// TwinCAT 3 PLC project tmo_optics
// Title: lcls-plc-tmo-optics
// Company: SLAC
// ProjectVersion: 0.0.0
// ProgramVersion: 3.1.4026.17
// CompilerDefines: K
// libraries:
//   LCLS General, * (SLAC)
//   lcls-twincat-common-components, * (SLAC)
//   lcls-twincat-optics, * (SLAC)
//   Tc2_MC2, * (Beckhoff Automation GmbH)
//   Tc2_SerialCom, * (Beckhoff Automation GmbH)
//   Tc2_Standard, * (Beckhoff Automation GmbH)
//   Tc2_System, * (Beckhoff Automation GmbH)
//   Tc2_Utilities, * (Beckhoff Automation GmbH)
//   Tc3_Module, * (Beckhoff Automation GmbH)
//   TcUnit, * (www.tcunit.org)
//   lcls-twincat-motion,4.4.0,SLAC
//   PMPS,3.12.0,SLAC - LCLS
// project tree:
//   DUTs/ ENUM_Si_B4C_Coating_States.TcDUT, ENUM_Si_B4C_Coating_States_1D.TcDUT, E_HomeState.TcDUT (not stored)
//   GVLs/ GVL_COM_Buffers.TcGVL (not stored), GVL_M1K4.TcGVL (not stored), GVL_M1K4_Constants.TcGVL (not stored), GVL_M2K4_RTD.TcGVL (not stored), GVL_M2K4_Constants.TcGVL (not stored), GVL_M3K4_RTD.TcGVL (not stored), GVL_M3K4_Constants.TcGVL (not stored), GVL_M4K4_RTD.TcGVL (not stored), GVL_M5K4_RTD.TcGVL (not stored), GVL_PMPS.TcGVL, GVL_SerialIO.TcGVL (not stored)
//   / PiezoDriver.TcTTO (not stored), PlcTask.TcTTO (not stored), SerialIO.TcTTO (not stored)
//   POUs/ FB_Offset_Coating_States.TcPOU (not stored), FB_KBO_Coating_States.TcPOU (not stored), Main.TcPOU, PRG_1_PlcTask.TcPOU (not stored), PRG_Environment.TcPOU (not stored), PRG_MR1K4_SOMS.TcPOU (not stored), PRG_MR2K4_KBO.TcPOU (not stored), PRG_MR3K4_KBO.TcPOU (not stored), PRG_MR4K4_KBO.TcPOU (not stored), PRG_MR5K4_KBO.TcPOU (not stored), PRG_PMPS.TcPOU, PRG_SL2K4_SCATTER.TcPOU (not stored), PRG_States.TcPOU, P_StripeProtections.TcPOU (not stored)
//   POUs/Serial Comm/ PiezoSerial.TcPOU (not stored), P_Serial_Com.TcPOU (not stored)
//   POUs/temp/ FB_SLITS.TcPOU (not stored)
// real-time tasks:
//   TASK PlcTask: cycle T#10ms, priority 20, ADS port 350
//   TASK PiezoDriver: cycle T#1ms, priority 3, ADS port 351
//   TASK SerialIO: cycle T#2ms, priority 1, ADS port 352
// motion (NC):
//   TASK NC-Task 1 SAF: cycle T#2ms, priority 4, ADS port 501
//   TASK NC-Task 1 SVB: cycle T#10ms, priority 8, ADS port 511
//   AXIS M1K4-Yup (id 1)
//   AXIS M1K4-Ydwn (id 2)
//   AXIS M1K4-Xup (id 3)
//   AXIS M1K4-Xdwn (id 4)
//   AXIS M1K4-Pitch (id 5)
//   AXIS M1K4-Bender (id 6)
//   AXIS M2K4-X (id 7)
//   AXIS M2K4-Y (id 8)
//   AXIS M2K4-rY (id 9)
//   AXIS M2K4-BEND-US (id 10)
//   AXIS M2K4-BEND-DS (id 11)
//   AXIS M3K4-X (id 12)
//   AXIS M3K4-Y (id 13)
//   AXIS M3K4-rX (id 14)
//   AXIS M3K4-BEND-US (id 15)
//   AXIS M3K4-BEND-DS (id 16)
//   AXIS M4K4 X (id 17)
//     Dynamic: AccelerationMaximum=100, DecelerationMaximum=100, Acceleration=100, Deceleration=100, DelayTime=0.008
//     Velo: Maximum=0.3
//     OtherSettings: AllowMotionCmdToSlave=true
//     encoder EncType=29
//       EncPara: ScaleFactorNumerator=5e-06, Offset=-28.961399, MaxCount=#xffffffff
//         SoftEndMinControl: Enable=true, Range=-11.4
//         SoftEndMaxControl: Enable=true, Range=13.4
//         Inc: RefSoftSyncMask=#x0000ffff
//     drive DrvType=24
//       DrvPara: Inverse=true
//         Analog: VeloReferenz=20, ScaleFactorActTorque=0.1
//         TimeComp: TaskDelayCycles=1
//     controller CtrType=2
//       CtrPara: PriorControlFactor=1
//         PosDiffControl: Range=0.2
//         PID: DeadBandPosition=0.001
//         Observer: BandWidth=20
//   AXIS M4K4 Y (id 18)
//     Dynamic: AccelerationMaximum=100, DecelerationMaximum=100, Acceleration=100, Deceleration=100, DelayTime=0.008
//     Velo: Maximum=0.2
//     OtherSettings: AllowMotionCmdToSlave=true
//     encoder EncType=29
//       EncPara: ScaleFactorNumerator=5e-06, Offset=-30.3992, MaxCount=#xffffffff
//         SoftEndMinControl: Enable=true, Range=-2.2
//         SoftEndMaxControl: Enable=true, Range=2.3
//         Inc: RefSoftSyncMask=#x0000ffff
//     drive DrvType=24
//       DrvPara: Inverse=true
//         Analog: VeloReferenz=1.25, ScaleFactorActTorque=0.1
//         TimeComp: TaskDelayCycles=1
//     controller CtrType=2
//       CtrPara: PriorControlFactor=1
//         PosDiffControl: Range=0.2
//         PID: PosKp=3, DeadBandPosition=0.001
//         Observer: BandWidth=20
//   AXIS M4K4 Z (id 19)
//     Dynamic: AccelerationMaximum=100, DecelerationMaximum=100, Acceleration=100, Deceleration=100, DelayTime=0.008
//     Velo: Maximum=0.2
//     OtherSettings: AllowMotionCmdToSlave=true
//     encoder EncType=29
//       EncPara: ScaleFactorNumerator=5e-06, Offset=-21445.3535, MaxCount=#xffffffff
//         SoftEndMinControl: Enable=true, Range=-1.5
//         SoftEndMaxControl: Enable=true, Range=0.85
//         Inc: RefSoftSyncMask=#x0000ffff
//     drive DrvType=24
//       DrvPara: Inverse=true
//         Analog: VeloReferenz=1.25, ScaleFactorActTorque=0.1
//         TimeComp: TaskDelayCycles=1
//     controller CtrType=2
//       CtrPara: PriorControlFactor=1
//         PosDiffControl: Range=0.2
//         PID: PosKp=2, DeadBandPosition=0.01
//         Observer: BandWidth=20
//   AXIS M4K4 rX (id 20)
//     General: UnitName=urad
//     Dynamic: AccelerationMaximum=100, DecelerationMaximum=100, Acceleration=100, Deceleration=100, DelayTime=0.008
//     Velo: Maximum=50
//     OtherSettings: AllowMotionCmdToSlave=true
//     encoder EncType=29
//       EncPara: ScaleFactorNumerator=0.0025826, Offset=-132192.8499, MaxCount=#xffffffff
//         FilterTime: TPos=0.2
//         SoftEndMinControl: Enable=true, Range=-500
//         SoftEndMaxControl: Enable=true, Range=500
//         Inc: RefSoftSyncMask=#x0000ffff
//     drive DrvType=24
//       Analog: VeloReferenz=140.69, ScaleFactorActTorque=0.1
//       TimeComp: TaskDelayCycles=1
//     controller CtrType=2
//       CtrPara: PriorControlFactor=1
//         PosDiffControl: Range=10
//         PID: PosExtKp=4, DeadBandPosition=0.01
//         Observer: BandWidth=20
//   AXIS M5K4 X (id 21)
//     Dynamic: AccelerationMaximum=100, DecelerationMaximum=100, Acceleration=100, Deceleration=100, DelayTime=0.008
//     Velo: Maximum=0.2
//     OtherSettings: AllowMotionCmdToSlave=true
//     encoder EncType=29
//       EncPara: ScaleFactorNumerator=5e-06, Offset=-29.80379, MaxCount=#xffffffff
//         SoftEndMinControl: Enable=true, Range=-2.1
//         SoftEndMaxControl: Enable=true, Range=2.6
//         Inc: RefSoftSyncMask=#x0000ffff
//     drive DrvType=24
//       DrvPara: Inverse=true
//         Analog: VeloReferenz=20, ScaleFactorActTorque=0.1
//         TimeComp: TaskDelayCycles=1
//     controller CtrType=2
//       CtrPara: PriorControlFactor=1
//         PosDiffControl: Range=0.2
//         PID: DeadBandPosition=0.001
//         Observer: BandWidth=20
//   AXIS M5K4 Y (id 22)
//     Dynamic: AccelerationMaximum=100, DecelerationMaximum=100, Acceleration=100, Deceleration=100, DelayTime=0.008
//     Velo: Maximum=0.3
//     OtherSettings: AllowMotionCmdToSlave=true
//     encoder EncType=29
//       EncPara: ScaleFactorNumerator=5e-06, Offset=-29.7766, MaxCount=#xffffffff
//         SoftEndMinControl: Enable=true, Range=-12.3
//         SoftEndMaxControl: Enable=true, Range=12.33
//         Inc: RefSoftSyncMask=#x0000ffff
//     drive DrvType=24
//       DrvPara: Inverse=true
//         Analog: VeloReferenz=1.25, ScaleFactorActTorque=0.1
//         TimeComp: TaskDelayCycles=1
//     controller CtrType=2
//       CtrPara: PriorControlFactor=1
//         PosDiffControl: Range=0.2
//         PID: DeadBandPosition=0.001
//         Observer: BandWidth=20
//   AXIS M5K4 Z (id 23)
//     Dynamic: AccelerationMaximum=100, DecelerationMaximum=100, Acceleration=100, Deceleration=100, DelayTime=0.008
//     Velo: Maximum=0.2
//     OtherSettings: AllowMotionCmdToSlave=true
//     encoder EncType=29
//       EncPara: ScaleFactorNumerator=5e-06, Offset=-21444.5039, MaxCount=#xffffffff
//         SoftEndMinControl: Enable=true, Range=-0.69
//         SoftEndMaxControl: Enable=true, Range=1.02
//         Inc: RefSoftSyncMask=#x0000ffff
//     drive DrvType=24
//       DrvPara: Inverse=true
//         Analog: VeloReferenz=1.25, ScaleFactorActTorque=0.1
//         TimeComp: TaskDelayCycles=1
//     controller CtrType=2
//       CtrPara: PriorControlFactor=1
//         PosDiffControl: Range=0.2
//         PID: PosExtVelo=1, DeadBandPosition=0.01
//         Observer: BandWidth=20
//   AXIS M5K4 rY (id 24)
//     General: UnitName=urad
//     Dynamic: AccelerationMaximum=100, DecelerationMaximum=100, Acceleration=100, Deceleration=100, DelayTime=0.008
//     Velo: Maximum=50
//     OtherSettings: AllowMotionCmdToSlave=true
//     encoder EncType=29
//       EncPara: ScaleFactorNumerator=0.00504, Offset=-198169.78, MaxCount=#xffffffff
//         FilterTime: TPos=0.2
//         SoftEndMinControl: Enable=true, Range=-500
//         SoftEndMaxControl: Enable=true, Range=500
//         Inc: RefSoftSyncMask=#x0000ffff
//     drive DrvType=24
//       Analog: VeloReferenz=192.31, ScaleFactorActTorque=0.1
//       TimeComp: TaskDelayCycles=1
//     controller CtrType=2
//       CtrPara: PriorControlFactor=1
//         PosDiffControl: Range=10
//         PID: PosKp=2, PosExtKp=10, DeadBandPosition=0.01
//         Observer: BandWidth=20
// I/O:
//   DEVICE Device 1 (EtherCAT)
// variable links:
//   Axes/M4K4 X <-> Device 1 (EtherCAT)/Term 1 (EK1200)/Term 39 (EK1122)/Term 94 (EK1100)/EL5042_M4K4X_M4K4Y
//     Enc/Inputs/In/nComState @bit 1 <-> WcState/InputToggle
//     Enc/Inputs/In/nComState <-> WcState/WcState
//     Enc/Inputs/In/nDataIn1 <-> FB Inputs Channel 1/Position
//     Enc/Inputs/In/nState1 @bit 12 <-> FB Inputs Channel 1/Status/Diag
//     Enc/Inputs/In/nState1 @bit 1 <-> FB Inputs Channel 1/Status/Error
//     Enc/Inputs/In/nState1 @bit 14 <-> FB Inputs Channel 1/Status/Input cycle counter
//     Enc/Inputs/In/nState1 @bit 2 <-> FB Inputs Channel 1/Status/Ready
//     Enc/Inputs/In/nState1 @bit 13 <-> FB Inputs Channel 1/Status/TxPDO State
//     Enc/Inputs/In/nState1 <-> FB Inputs Channel 1/Status/Warning
//   Axes/M4K4 X <-> Device 1 (EtherCAT)/Term 1 (EK1200)/Term 39 (EK1122)/Term 94 (EK1100)/EL7041-0052_M4K4X
//     Drive/Inputs/In/nState1 @bit 3 <-> STM Status/Status/Error
//     Drive/Inputs/In/nState1 @bit 5 <-> STM Status/Status/Moving negative
//     Drive/Inputs/In/nState1 @bit 4 <-> STM Status/Status/Moving positive
//     Drive/Inputs/In/nState1 @bit 1 <-> STM Status/Status/Ready
//     Drive/Inputs/In/nState1 <-> STM Status/Status/Ready to enable
//     Drive/Inputs/In/nState1 @bit 6 <-> STM Status/Status/Torque reduced
//     Drive/Inputs/In/nState1 @bit 2 <-> STM Status/Status/Warning
//     Drive/Inputs/In/nState2 @bit 3 <-> STM Status/Status/Digital input 1
//     Drive/Inputs/In/nState2 @bit 4 <-> STM Status/Status/Digital input 2
//     Drive/Inputs/In/nState2 @bit 5 <-> STM Status/Status/Sync error
//     Drive/Inputs/In/nState2 @bit 7 <-> STM Status/Status/TxPDO Toggle
//     Drive/Inputs/In/nState4 @bit 1 <-> WcState/InputToggle
//     Drive/Inputs/In/nState4 <-> WcState/WcState
//     Drive/Outputs/Out/nCtrl1 <-> STM Control/Control/Enable
//     Drive/Outputs/Out/nCtrl1 @bit 2 <-> STM Control/Control/Reduce torque
//     Drive/Outputs/Out/nCtrl1 @bit 1 <-> STM Control/Control/Reset
//     Drive/Outputs/Out/nDataOut2[0] <-> STM Velocity/Velocity
//   Axes/M4K4 Y <-> Device 1 (EtherCAT)/Term 1 (EK1200)/Term 39 (EK1122)/Term 94 (EK1100)/EL5042_M4K4X_M4K4Y
//     Enc/Inputs/In/nComState @bit 1 <-> WcState/InputToggle
//     Enc/Inputs/In/nComState <-> WcState/WcState
//     Enc/Inputs/In/nDataIn1 <-> FB Inputs Channel 2/Position
//     Enc/Inputs/In/nState1 @bit 12 <-> FB Inputs Channel 2/Status/Diag
//     Enc/Inputs/In/nState1 @bit 1 <-> FB Inputs Channel 2/Status/Error
//     Enc/Inputs/In/nState1 @bit 14 <-> FB Inputs Channel 2/Status/Input cycle counter
//     Enc/Inputs/In/nState1 @bit 2 <-> FB Inputs Channel 2/Status/Ready
//     Enc/Inputs/In/nState1 @bit 13 <-> FB Inputs Channel 2/Status/TxPDO State
//     Enc/Inputs/In/nState1 <-> FB Inputs Channel 2/Status/Warning
//   Axes/M4K4 Y <-> Device 1 (EtherCAT)/Term 1 (EK1200)/Term 39 (EK1122)/Term 94 (EK1100)/EL7041-0052_M4K4Y
//     Drive/Inputs/In/nState1 @bit 3 <-> STM Status/Status/Error
//     Drive/Inputs/In/nState1 @bit 5 <-> STM Status/Status/Moving negative
//     Drive/Inputs/In/nState1 @bit 4 <-> STM Status/Status/Moving positive
//     Drive/Inputs/In/nState1 @bit 1 <-> STM Status/Status/Ready
//     Drive/Inputs/In/nState1 <-> STM Status/Status/Ready to enable
//     Drive/Inputs/In/nState1 @bit 6 <-> STM Status/Status/Torque reduced
//     Drive/Inputs/In/nState1 @bit 2 <-> STM Status/Status/Warning
//     Drive/Inputs/In/nState2 @bit 3 <-> STM Status/Status/Digital input 1
//     Drive/Inputs/In/nState2 @bit 4 <-> STM Status/Status/Digital input 2
//     Drive/Inputs/In/nState2 @bit 5 <-> STM Status/Status/Sync error
//     Drive/Inputs/In/nState2 @bit 7 <-> STM Status/Status/TxPDO Toggle
//     Drive/Inputs/In/nState4 @bit 1 <-> WcState/InputToggle
//     Drive/Inputs/In/nState4 <-> WcState/WcState
//     Drive/Outputs/Out/nCtrl1 <-> STM Control/Control/Enable
//     Drive/Outputs/Out/nCtrl1 @bit 2 <-> STM Control/Control/Reduce torque
//     Drive/Outputs/Out/nCtrl1 @bit 1 <-> STM Control/Control/Reset
//     Drive/Outputs/Out/nDataOut2[0] <-> STM Velocity/Velocity
//   Axes/M4K4 Z <-> Device 1 (EtherCAT)/Term 1 (EK1200)/Term 39 (EK1122)/Term 94 (EK1100)/EL5042_M4K4Z_M4K4rX
//     Enc/Inputs/In/nComState @bit 1 <-> WcState/InputToggle
//     Enc/Inputs/In/nComState <-> WcState/WcState
//     Enc/Inputs/In/nDataIn1 <-> FB Inputs Channel 1/Position
//     Enc/Inputs/In/nState1 @bit 12 <-> FB Inputs Channel 1/Status/Diag
//     Enc/Inputs/In/nState1 @bit 1 <-> FB Inputs Channel 1/Status/Error
//     Enc/Inputs/In/nState1 @bit 14 <-> FB Inputs Channel 1/Status/Input cycle counter
//     Enc/Inputs/In/nState1 @bit 2 <-> FB Inputs Channel 1/Status/Ready
//     Enc/Inputs/In/nState1 @bit 13 <-> FB Inputs Channel 1/Status/TxPDO State
//     Enc/Inputs/In/nState1 <-> FB Inputs Channel 1/Status/Warning
//   Axes/M4K4 Z <-> Device 1 (EtherCAT)/Term 1 (EK1200)/Term 39 (EK1122)/Term 94 (EK1100)/EL7041-0052_M4K4Z
//     Drive/Inputs/In/nState1 @bit 3 <-> STM Status/Status/Error
//     Drive/Inputs/In/nState1 @bit 5 <-> STM Status/Status/Moving negative
//     Drive/Inputs/In/nState1 @bit 4 <-> STM Status/Status/Moving positive
//     Drive/Inputs/In/nState1 @bit 1 <-> STM Status/Status/Ready
//     Drive/Inputs/In/nState1 <-> STM Status/Status/Ready to enable
//     Drive/Inputs/In/nState1 @bit 6 <-> STM Status/Status/Torque reduced
//     Drive/Inputs/In/nState1 @bit 2 <-> STM Status/Status/Warning
//     Drive/Inputs/In/nState2 @bit 3 <-> STM Status/Status/Digital input 1
//     Drive/Inputs/In/nState2 @bit 4 <-> STM Status/Status/Digital input 2
//     Drive/Inputs/In/nState2 @bit 5 <-> STM Status/Status/Sync error
//     Drive/Inputs/In/nState2 @bit 7 <-> STM Status/Status/TxPDO Toggle
//     Drive/Inputs/In/nState4 @bit 1 <-> WcState/InputToggle
//     Drive/Inputs/In/nState4 <-> WcState/WcState
//     Drive/Outputs/Out/nCtrl1 <-> STM Control/Control/Enable
//     Drive/Outputs/Out/nCtrl1 @bit 2 <-> STM Control/Control/Reduce torque
//     Drive/Outputs/Out/nCtrl1 @bit 1 <-> STM Control/Control/Reset
//     Drive/Outputs/Out/nDataOut2[0] <-> STM Velocity/Velocity
//   Axes/M4K4 rX <-> Device 1 (EtherCAT)/Term 1 (EK1200)/Term 39 (EK1122)/Term 94 (EK1100)/EL5042_M4K4Z_M4K4rX
//     Enc/Inputs/In/nComState @bit 1 <-> WcState/InputToggle
//     Enc/Inputs/In/nComState <-> WcState/WcState
//     Enc/Inputs/In/nDataIn1 <-> FB Inputs Channel 2/Position
//     Enc/Inputs/In/nState1 @bit 12 <-> FB Inputs Channel 2/Status/Diag
//     Enc/Inputs/In/nState1 @bit 1 <-> FB Inputs Channel 2/Status/Error
//     Enc/Inputs/In/nState1 @bit 14 <-> FB Inputs Channel 2/Status/Input cycle counter
//     Enc/Inputs/In/nState1 @bit 2 <-> FB Inputs Channel 2/Status/Ready
//     Enc/Inputs/In/nState1 @bit 13 <-> FB Inputs Channel 2/Status/TxPDO State
//     Enc/Inputs/In/nState1 <-> FB Inputs Channel 2/Status/Warning
//   Axes/M4K4 rX <-> Device 1 (EtherCAT)/Term 1 (EK1200)/Term 39 (EK1122)/Term 94 (EK1100)/EL7041-0052_M4K4rX
//     Drive/Inputs/In/nState1 @bit 3 <-> STM Status/Status/Error
//     Drive/Inputs/In/nState1 @bit 5 <-> STM Status/Status/Moving negative
//     Drive/Inputs/In/nState1 @bit 4 <-> STM Status/Status/Moving positive
//     Drive/Inputs/In/nState1 @bit 1 <-> STM Status/Status/Ready
//     Drive/Inputs/In/nState1 <-> STM Status/Status/Ready to enable
//     Drive/Inputs/In/nState1 @bit 6 <-> STM Status/Status/Torque reduced
//     Drive/Inputs/In/nState1 @bit 2 <-> STM Status/Status/Warning
//     Drive/Inputs/In/nState2 @bit 3 <-> STM Status/Status/Digital input 1
//     Drive/Inputs/In/nState2 @bit 4 <-> STM Status/Status/Digital input 2
//     Drive/Inputs/In/nState2 @bit 5 <-> STM Status/Status/Sync error
//     Drive/Inputs/In/nState2 @bit 7 <-> STM Status/Status/TxPDO Toggle
//     Drive/Inputs/In/nState4 @bit 1 <-> WcState/InputToggle
//     Drive/Inputs/In/nState4 <-> WcState/WcState
//     Drive/Outputs/Out/nCtrl1 <-> STM Control/Control/Enable
//     Drive/Outputs/Out/nCtrl1 @bit 2 <-> STM Control/Control/Reduce torque
//     Drive/Outputs/Out/nCtrl1 @bit 1 <-> STM Control/Control/Reset
//     Drive/Outputs/Out/nDataOut2[0] <-> STM Velocity/Velocity
//   Axes/M5K4 X <-> Device 1 (EtherCAT)/Term 1 (EK1200)/Term 39 (EK1122)/Term 94 (EK1100)/EL5042_M5K4X_M5K4Y
//     Enc/Inputs/In/nComState @bit 1 <-> WcState/InputToggle
//     Enc/Inputs/In/nComState <-> WcState/WcState
//     Enc/Inputs/In/nDataIn1 <-> FB Inputs Channel 1/Position
//     Enc/Inputs/In/nState1 @bit 12 <-> FB Inputs Channel 1/Status/Diag
//     Enc/Inputs/In/nState1 @bit 1 <-> FB Inputs Channel 1/Status/Error
//     Enc/Inputs/In/nState1 @bit 14 <-> FB Inputs Channel 1/Status/Input cycle counter
//     Enc/Inputs/In/nState1 @bit 2 <-> FB Inputs Channel 1/Status/Ready
//     Enc/Inputs/In/nState1 @bit 13 <-> FB Inputs Channel 1/Status/TxPDO State
//     Enc/Inputs/In/nState1 <-> FB Inputs Channel 1/Status/Warning
//   Axes/M5K4 X <-> Device 1 (EtherCAT)/Term 1 (EK1200)/Term 39 (EK1122)/Term 94 (EK1100)/EL7041-0052_M5K4X
//     Drive/Inputs/In/nState1 @bit 3 <-> STM Status/Status/Error
//     Drive/Inputs/In/nState1 @bit 5 <-> STM Status/Status/Moving negative
//     Drive/Inputs/In/nState1 @bit 4 <-> STM Status/Status/Moving positive
//     Drive/Inputs/In/nState1 @bit 1 <-> STM Status/Status/Ready
//     Drive/Inputs/In/nState1 <-> STM Status/Status/Ready to enable
//     Drive/Inputs/In/nState1 @bit 6 <-> STM Status/Status/Torque reduced
//     Drive/Inputs/In/nState1 @bit 2 <-> STM Status/Status/Warning
//     Drive/Inputs/In/nState2 @bit 3 <-> STM Status/Status/Digital input 1
//     Drive/Inputs/In/nState2 @bit 4 <-> STM Status/Status/Digital input 2
//     Drive/Inputs/In/nState2 @bit 5 <-> STM Status/Status/Sync error
//     Drive/Inputs/In/nState2 @bit 7 <-> STM Status/Status/TxPDO Toggle
//     Drive/Inputs/In/nState4 @bit 1 <-> WcState/InputToggle
//     Drive/Inputs/In/nState4 <-> WcState/WcState
//     Drive/Outputs/Out/nCtrl1 <-> STM Control/Control/Enable
//     Drive/Outputs/Out/nCtrl1 @bit 2 <-> STM Control/Control/Reduce torque
//     Drive/Outputs/Out/nCtrl1 @bit 1 <-> STM Control/Control/Reset
//     Drive/Outputs/Out/nDataOut2[0] <-> STM Velocity/Velocity
//   Axes/M5K4 Y <-> Device 1 (EtherCAT)/Term 1 (EK1200)/Term 39 (EK1122)/Term 94 (EK1100)/EL5042_M5K4X_M5K4Y
//     Enc/Inputs/In/nComState @bit 1 <-> WcState/InputToggle
//     Enc/Inputs/In/nComState <-> WcState/WcState
//     Enc/Inputs/In/nDataIn1 <-> FB Inputs Channel 2/Position
//     Enc/Inputs/In/nState1 @bit 12 <-> FB Inputs Channel 2/Status/Diag
//     Enc/Inputs/In/nState1 @bit 1 <-> FB Inputs Channel 2/Status/Error
//     Enc/Inputs/In/nState1 @bit 14 <-> FB Inputs Channel 2/Status/Input cycle counter
//     Enc/Inputs/In/nState1 @bit 2 <-> FB Inputs Channel 2/Status/Ready
//     Enc/Inputs/In/nState1 @bit 13 <-> FB Inputs Channel 2/Status/TxPDO State
//     Enc/Inputs/In/nState1 <-> FB Inputs Channel 2/Status/Warning
//   Axes/M5K4 Y <-> Device 1 (EtherCAT)/Term 1 (EK1200)/Term 39 (EK1122)/Term 94 (EK1100)/EL7041-0052_M5K4Y
//     Drive/Inputs/In/nState1 @bit 3 <-> STM Status/Status/Error
//     Drive/Inputs/In/nState1 @bit 5 <-> STM Status/Status/Moving negative
//     Drive/Inputs/In/nState1 @bit 4 <-> STM Status/Status/Moving positive
//     Drive/Inputs/In/nState1 @bit 1 <-> STM Status/Status/Ready
//     Drive/Inputs/In/nState1 <-> STM Status/Status/Ready to enable
//     Drive/Inputs/In/nState1 @bit 6 <-> STM Status/Status/Torque reduced
//     Drive/Inputs/In/nState1 @bit 2 <-> STM Status/Status/Warning
//     Drive/Inputs/In/nState2 @bit 3 <-> STM Status/Status/Digital input 1
//     Drive/Inputs/In/nState2 @bit 4 <-> STM Status/Status/Digital input 2
//     Drive/Inputs/In/nState2 @bit 5 <-> STM Status/Status/Sync error
//     Drive/Inputs/In/nState2 @bit 7 <-> STM Status/Status/TxPDO Toggle
//     Drive/Inputs/In/nState4 @bit 1 <-> WcState/InputToggle
//     Drive/Inputs/In/nState4 <-> WcState/WcState
//     Drive/Outputs/Out/nCtrl1 <-> STM Control/Control/Enable
//     Drive/Outputs/Out/nCtrl1 @bit 2 <-> STM Control/Control/Reduce torque
//     Drive/Outputs/Out/nCtrl1 @bit 1 <-> STM Control/Control/Reset
//     Drive/Outputs/Out/nDataOut2[0] <-> STM Velocity/Velocity
//   Axes/M5K4 Z <-> Device 1 (EtherCAT)/Term 1 (EK1200)/Term 39 (EK1122)/Term 94 (EK1100)/EL5042_M5K4Z_M5K4rY
//     Enc/Inputs/In/nComState @bit 1 <-> WcState/InputToggle
//     Enc/Inputs/In/nComState <-> WcState/WcState
//     Enc/Inputs/In/nDataIn1 <-> FB Inputs Channel 1/Position
//     Enc/Inputs/In/nState1 @bit 12 <-> FB Inputs Channel 1/Status/Diag
//     Enc/Inputs/In/nState1 @bit 1 <-> FB Inputs Channel 1/Status/Error
//     Enc/Inputs/In/nState1 @bit 14 <-> FB Inputs Channel 1/Status/Input cycle counter
//     Enc/Inputs/In/nState1 @bit 2 <-> FB Inputs Channel 1/Status/Ready
//     Enc/Inputs/In/nState1 @bit 13 <-> FB Inputs Channel 1/Status/TxPDO State
//     Enc/Inputs/In/nState1 <-> FB Inputs Channel 1/Status/Warning
//   Axes/M5K4 Z <-> Device 1 (EtherCAT)/Term 1 (EK1200)/Term 39 (EK1122)/Term 94 (EK1100)/EL7041-0052_M5K4Z
//     Drive/Inputs/In/nState1 @bit 3 <-> STM Status/Status/Error
//     Drive/Inputs/In/nState1 @bit 5 <-> STM Status/Status/Moving negative
//     Drive/Inputs/In/nState1 @bit 4 <-> STM Status/Status/Moving positive
//     Drive/Inputs/In/nState1 @bit 1 <-> STM Status/Status/Ready
//     Drive/Inputs/In/nState1 <-> STM Status/Status/Ready to enable
//     Drive/Inputs/In/nState1 @bit 6 <-> STM Status/Status/Torque reduced
//     Drive/Inputs/In/nState1 @bit 2 <-> STM Status/Status/Warning
//     Drive/Inputs/In/nState2 @bit 3 <-> STM Status/Status/Digital input 1
//     Drive/Inputs/In/nState2 @bit 4 <-> STM Status/Status/Digital input 2
//     Drive/Inputs/In/nState2 @bit 5 <-> STM Status/Status/Sync error
//     Drive/Inputs/In/nState2 @bit 7 <-> STM Status/Status/TxPDO Toggle
//     Drive/Inputs/In/nState4 @bit 1 <-> WcState/InputToggle
//     Drive/Inputs/In/nState4 <-> WcState/WcState
//     Drive/Outputs/Out/nCtrl1 <-> STM Control/Control/Enable
//     Drive/Outputs/Out/nCtrl1 @bit 2 <-> STM Control/Control/Reduce torque
//     Drive/Outputs/Out/nCtrl1 @bit 1 <-> STM Control/Control/Reset
//     Drive/Outputs/Out/nDataOut2[0] <-> STM Velocity/Velocity
//   Axes/M5K4 rY <-> Device 1 (EtherCAT)/Term 1 (EK1200)/Term 39 (EK1122)/Term 94 (EK1100)/EL5042_M5K4Z_M5K4rY
//     Enc/Inputs/In/nComState @bit 1 <-> WcState/InputToggle
//     Enc/Inputs/In/nComState <-> WcState/WcState
//     Enc/Inputs/In/nDataIn1 <-> FB Inputs Channel 2/Position
//     Enc/Inputs/In/nState1 @bit 12 <-> FB Inputs Channel 2/Status/Diag
//     Enc/Inputs/In/nState1 @bit 1 <-> FB Inputs Channel 2/Status/Error
//     Enc/Inputs/In/nState1 @bit 14 <-> FB Inputs Channel 2/Status/Input cycle counter
//     Enc/Inputs/In/nState1 @bit 2 <-> FB Inputs Channel 2/Status/Ready
//     Enc/Inputs/In/nState1 @bit 13 <-> FB Inputs Channel 2/Status/TxPDO State
//     Enc/Inputs/In/nState1 <-> FB Inputs Channel 2/Status/Warning
//   Axes/M5K4 rY <-> Device 1 (EtherCAT)/Term 1 (EK1200)/Term 39 (EK1122)/Term 94 (EK1100)/EL7041-0052_M5K4rY
//     Drive/Inputs/In/nState1 @bit 3 <-> STM Status/Status/Error
//     Drive/Inputs/In/nState1 @bit 5 <-> STM Status/Status/Moving negative
//     Drive/Inputs/In/nState1 @bit 4 <-> STM Status/Status/Moving positive
//     Drive/Inputs/In/nState1 @bit 1 <-> STM Status/Status/Ready
//     Drive/Inputs/In/nState1 <-> STM Status/Status/Ready to enable
//     Drive/Inputs/In/nState1 @bit 6 <-> STM Status/Status/Torque reduced
//     Drive/Inputs/In/nState1 @bit 2 <-> STM Status/Status/Warning
//     Drive/Inputs/In/nState2 @bit 3 <-> STM Status/Status/Digital input 1
//     Drive/Inputs/In/nState2 @bit 4 <-> STM Status/Status/Digital input 2
//     Drive/Inputs/In/nState2 @bit 5 <-> STM Status/Status/Sync error
//     Drive/Inputs/In/nState2 @bit 7 <-> STM Status/Status/TxPDO Toggle
//     Drive/Inputs/In/nState4 @bit 1 <-> WcState/InputToggle
//     Drive/Inputs/In/nState4 <-> WcState/WcState
//     Drive/Outputs/Out/nCtrl1 <-> STM Control/Control/Enable
//     Drive/Outputs/Out/nCtrl1 @bit 2 <-> STM Control/Control/Reduce torque
//     Drive/Outputs/Out/nCtrl1 @bit 1 <-> STM Control/Control/Reset
//     Drive/Outputs/Out/nDataOut2[0] <-> STM Velocity/Velocity
//   tmo_optics Instance <-> Device 1 (EtherCAT)/Term 1 (EK1200)/PMPS_FFO
//     PlcTask Outputs/GVL_PMPS.g_FastFaultOutput1.q_xFastFaultOut <-> Channel 1/Output
//     PlcTask Outputs/GVL_PMPS.g_FastFaultOutput2.q_xFastFaultOut <-> Channel 2/Output
//   tmo_optics Instance <-> Device 1 (EtherCAT)/Term 1 (EK1200)/PMPS_PRE
//     PlcTask Inputs/PRG_PMPS.fbArbiterIO.i_stCurrentBP <-> IO Inputs/CurrentBP
//     PlcTask Inputs/PRG_PMPS.fbArbiterIO.xTxPDO_state <-> SYNC Inputs/TxPDO state
//     PlcTask Inputs/PRG_PMPS.fbArbiterIO.xTxPDO_toggle <-> SYNC Inputs/TxPDO toggle
//     PlcTask Outputs/PRG_PMPS.fbArbiterIO.q_stRequestedBP <-> IO Outputs/RequestedBP
//   tmo_optics Instance <-> Device 1 (EtherCAT)/Term 1 (EK1200)/Term 39 (EK1122)/B940-009-R19-DRL-04 (EK1100)/SL2K4-EL5072-E1
//     PlcTask Inputs/Main.M25.nRawEncoderDINT <-> IND Inputs Channel 1/Position
//     PlcTask Inputs/Main.M26.nRawEncoderDINT <-> IND Inputs Channel 2/Position
//   tmo_optics Instance <-> Device 1 (EtherCAT)/Term 1 (EK1200)/Term 39 (EK1122)/B940-009-R19-DRL-04 (EK1100)/SL2K4-EL5072-E2
//     PlcTask Inputs/Main.M27.nRawEncoderDINT <-> IND Inputs Channel 1/Position
//     PlcTask Inputs/Main.M28.nRawEncoderDINT <-> IND Inputs Channel 2/Position
//   tmo_optics Instance <-> Device 1 (EtherCAT)/Term 1 (EK1200)/Term 39 (EK1122)/Term 110 (EK1100)/EL3054_FWM_PRSM_MR45K4
//     PlcTask Inputs/PRG_MR4K4_KBO.fbCoolingPanel.fbFlow_1.iRaw <-> AI Standard Channel 1/Value
//     PlcTask Inputs/PRG_MR5K4_KBO.fbCoolingPanel.fbFlow_1.iRaw <-> AI Standard Channel 3/Value
//     PlcTask Inputs/PRG_MR4K4_KBO.fbCoolingPanel.fbPress_1.iRaw <-> AI Standard Channel 2/Value
//     PlcTask Inputs/PRG_MR5K4_KBO.fbCoolingPanel.fbPress_1.iRaw <-> AI Standard Channel 2/Value
//   tmo_optics Instance <-> Device 1 (EtherCAT)/Term 1 (EK1200)/Term 39 (EK1122)/Term 110 (EK1100)/EL3204_M4K4
//     PlcTask Inputs/GVL_M4K4_RTD.nM4K4_Chin_Left_RTD.bError <-> RTD Inputs Channel 1/Status/Error
//     PlcTask Inputs/GVL_M4K4_RTD.nM4K4_Chin_Left_RTD.bOverrange <-> RTD Inputs Channel 1/Status/Overrange
//     PlcTask Inputs/GVL_M4K4_RTD.nM4K4_Chin_Left_RTD.bUnderrange <-> RTD Inputs Channel 1/Status/Underrange
//     PlcTask Inputs/GVL_M4K4_RTD.nM4K4_Chin_Left_RTD.iRaw <-> RTD Inputs Channel 1/Value
//     PlcTask Inputs/GVL_M4K4_RTD.nM4K4_Chin_Right_RTD.bError <-> RTD Inputs Channel 2/Status/Error
//     PlcTask Inputs/GVL_M4K4_RTD.nM4K4_Chin_Right_RTD.bOverrange <-> RTD Inputs Channel 2/Status/Overrange
//     PlcTask Inputs/GVL_M4K4_RTD.nM4K4_Chin_Right_RTD.bUnderrange <-> RTD Inputs Channel 2/Status/Underrange
//     PlcTask Inputs/GVL_M4K4_RTD.nM4K4_Chin_Right_RTD.iRaw <-> RTD Inputs Channel 2/Value
//     PlcTask Inputs/GVL_M4K4_RTD.nM4K4_Chin_Tail_RTD.bError <-> RTD Inputs Channel 3/Status/Error
//     PlcTask Inputs/GVL_M4K4_RTD.nM4K4_Chin_Tail_RTD.bOverrange <-> RTD Inputs Channel 3/Status/Overrange
//     PlcTask Inputs/GVL_M4K4_RTD.nM4K4_Chin_Tail_RTD.bUnderrange <-> RTD Inputs Channel 3/Status/Underrange
//     PlcTask Inputs/GVL_M4K4_RTD.nM4K4_Chin_Tail_RTD.iRaw <-> RTD Inputs Channel 3/Value
//   tmo_optics Instance <-> Device 1 (EtherCAT)/Term 1 (EK1200)/Term 39 (EK1122)/Term 110 (EK1100)/EL3204_M5K4
//     PlcTask Inputs/GVL_M5K4_RTD.nM5K4_Chin_Left_RTD.bError <-> RTD Inputs Channel 1/Status/Error
//     PlcTask Inputs/GVL_M5K4_RTD.nM5K4_Chin_Left_RTD.bOverrange <-> RTD Inputs Channel 1/Status/Overrange
//     PlcTask Inputs/GVL_M5K4_RTD.nM5K4_Chin_Left_RTD.bUnderrange <-> RTD Inputs Channel 1/Status/Underrange
//     PlcTask Inputs/GVL_M5K4_RTD.nM5K4_Chin_Left_RTD.iRaw <-> RTD Inputs Channel 1/Value
//     PlcTask Inputs/GVL_M5K4_RTD.nM5K4_Chin_Right_RTD.bError <-> RTD Inputs Channel 2/Status/Error
//     PlcTask Inputs/GVL_M5K4_RTD.nM5K4_Chin_Right_RTD.bOverrange <-> RTD Inputs Channel 2/Status/Overrange
//     PlcTask Inputs/GVL_M5K4_RTD.nM5K4_Chin_Right_RTD.bUnderrange <-> RTD Inputs Channel 2/Status/Underrange
//     PlcTask Inputs/GVL_M5K4_RTD.nM5K4_Chin_Right_RTD.iRaw <-> RTD Inputs Channel 2/Value
//     PlcTask Inputs/GVL_M5K4_RTD.nM5K4_Chin_Tail_RTD.bError <-> RTD Inputs Channel 3/Status/Error
//     PlcTask Inputs/GVL_M5K4_RTD.nM5K4_Chin_Tail_RTD.bOverrange <-> RTD Inputs Channel 3/Status/Overrange
//     PlcTask Inputs/GVL_M5K4_RTD.nM5K4_Chin_Tail_RTD.bUnderrange <-> RTD Inputs Channel 3/Status/Underrange
//     PlcTask Inputs/GVL_M5K4_RTD.nM5K4_Chin_Tail_RTD.iRaw <-> RTD Inputs Channel 3/Value
//   tmo_optics Instance <-> Device 1 (EtherCAT)/Term 1 (EK1200)/Term 39 (EK1122)/Term 94 (EK1100)/EL5042_M4K4X_M4K4Y
//     PlcTask Inputs/Main.M17.nRawEncoderULINT <-> FB Inputs Channel 1/Position
//     PlcTask Inputs/Main.M18.nRawEncoderULINT <-> FB Inputs Channel 2/Position
//   tmo_optics Instance <-> Device 1 (EtherCAT)/Term 1 (EK1200)/Term 39 (EK1122)/Term 94 (EK1100)/EL5042_M4K4Z_M4K4rX
//     PlcTask Inputs/Main.M19.nRawEncoderULINT <-> FB Inputs Channel 1/Position
//     PlcTask Inputs/Main.M20.nRawEncoderULINT <-> FB Inputs Channel 2/Position
//   tmo_optics Instance <-> Device 1 (EtherCAT)/Term 1 (EK1200)/Term 39 (EK1122)/Term 94 (EK1100)/EL5042_M5K4X_M5K4Y
//     PlcTask Inputs/Main.M21.nRawEncoderULINT <-> FB Inputs Channel 1/Position
//     PlcTask Inputs/Main.M22.nRawEncoderULINT <-> FB Inputs Channel 2/Position
//   tmo_optics Instance <-> Device 1 (EtherCAT)/Term 1 (EK1200)/Term 39 (EK1122)/Term 94 (EK1100)/EL5042_M5K4Z_M5K4rY
//     PlcTask Inputs/Main.M23.nRawEncoderULINT <-> FB Inputs Channel 1/Position
//     PlcTask Inputs/Main.M24.nRawEncoderULINT <-> FB Inputs Channel 2/Position
//   tmo_optics Instance <-> Device 1 (EtherCAT)/Term 1 (EK1200)/Term 39 (EK1122)/Term 94 (EK1100)/EL7041-0052_M4K4X
//     PlcTask Inputs/Main.M17.bLimitBackwardEnable <-> STM Status/Status/Digital input 2
//     PlcTask Inputs/Main.M17.bLimitForwardEnable <-> STM Status/Status/Digital input 1
//   tmo_optics Instance <-> Device 1 (EtherCAT)/Term 1 (EK1200)/Term 39 (EK1122)/Term 94 (EK1100)/EL7041-0052_M4K4Y
//     PlcTask Inputs/Main.M18.bLimitBackwardEnable <-> STM Status/Status/Digital input 2
//     PlcTask Inputs/Main.M18.bLimitForwardEnable <-> STM Status/Status/Digital input 1
//   tmo_optics Instance <-> Device 1 (EtherCAT)/Term 1 (EK1200)/Term 39 (EK1122)/Term 94 (EK1100)/EL7041-0052_M4K4Z
//     PlcTask Inputs/Main.M19.bLimitBackwardEnable <-> STM Status/Status/Digital input 1
//     PlcTask Inputs/Main.M19.bLimitForwardEnable <-> STM Status/Status/Digital input 2
//   tmo_optics Instance <-> Device 1 (EtherCAT)/Term 1 (EK1200)/Term 39 (EK1122)/Term 94 (EK1100)/EL7041-0052_M4K4rX
//     PlcTask Inputs/Main.M20.bLimitBackwardEnable <-> STM Status/Status/Digital input 2
//     PlcTask Inputs/Main.M20.bLimitForwardEnable <-> STM Status/Status/Digital input 1
//   tmo_optics Instance <-> Device 1 (EtherCAT)/Term 1 (EK1200)/Term 39 (EK1122)/Term 94 (EK1100)/EL7041-0052_M5K4X
//     PlcTask Inputs/Main.M21.bLimitBackwardEnable <-> STM Status/Status/Digital input 2
//     PlcTask Inputs/Main.M21.bLimitForwardEnable <-> STM Status/Status/Digital input 1
//   tmo_optics Instance <-> Device 1 (EtherCAT)/Term 1 (EK1200)/Term 39 (EK1122)/Term 94 (EK1100)/EL7041-0052_M5K4Y
//     PlcTask Inputs/Main.M22.bLimitBackwardEnable <-> STM Status/Status/Digital input 2
//     PlcTask Inputs/Main.M22.bLimitForwardEnable <-> STM Status/Status/Digital input 1
//   tmo_optics Instance <-> Device 1 (EtherCAT)/Term 1 (EK1200)/Term 39 (EK1122)/Term 94 (EK1100)/EL7041-0052_M5K4Z
//     PlcTask Inputs/Main.M23.bLimitBackwardEnable <-> STM Status/Status/Digital input 1
//     PlcTask Inputs/Main.M23.bLimitForwardEnable <-> STM Status/Status/Digital input 2
//   tmo_optics Instance <-> Device 1 (EtherCAT)/Term 1 (EK1200)/Term 39 (EK1122)/Term 94 (EK1100)/EL7041-0052_M5K4rY
//     PlcTask Inputs/Main.M24.bLimitBackwardEnable <-> STM Status/Status/Digital input 2
//     PlcTask Inputs/Main.M24.bLimitForwardEnable <-> STM Status/Status/Digital input 1
//   tmo_optics Instance <-> Device 1 (EtherCAT)/Term 1 (EK1200)/Term 39 (EK1122)/Term 94 (EK1100)/Term 109 (EL1004)
//     PlcTask Inputs/Main.bDreamEnable1 <-> Channel 1/Input
//     PlcTask Inputs/Main.bDreamEnable2 <-> Channel 2/Input
//   tmo_optics Instance <-> Device 1 (EtherCAT)/Term 1 (EK1200)/Term 5 (EK1122)/EP2008-0001_M1K4_VCV
//     PlcTask Outputs/PRG_MR1K4_SOMS.bActivateVarCool <-> Channel 1/Output
//   tmo_optics Instance <-> Device 1 (EtherCAT)/Term 1 (EK1200)/Term 5 (EK1122)/Term 20 (EK1100)/EL1004_M2K4_M3K4_STO
//     PlcTask Inputs/Main.LAMPbSTOEnable1 <-> Channel 1/Input
//     PlcTask Inputs/Main.LAMPbSTOEnable2 <-> Channel 2/Input
//   tmo_optics Instance <-> Device 1 (EtherCAT)/Term 1 (EK1200)/Term 5 (EK1122)/Term 20 (EK1100)/EL5042_M2K4X_M2K4Y
//     PlcTask Inputs/Main.M7.nRawEncoderULINT <-> FB Inputs Channel 1/Position
//     PlcTask Inputs/Main.M8.nRawEncoderULINT <-> FB Inputs Channel 2/Position
//   tmo_optics Instance <-> Device 1 (EtherCAT)/Term 1 (EK1200)/Term 5 (EK1122)/Term 20 (EK1100)/EL5042_M2K4_BEND_USDS
//     PlcTask Inputs/Main.M10.nRawEncoderULINT <-> FB Inputs Channel 1/Position
//     PlcTask Inputs/Main.M11.nRawEncoderULINT <-> FB Inputs Channel 2/Position
//     PlcTask Inputs/Main.M16.nRawEncoderULINT <-> FB Inputs Channel 2/Position
//   tmo_optics Instance <-> Device 1 (EtherCAT)/Term 1 (EK1200)/Term 5 (EK1122)/Term 20 (EK1100)/EL5042_M2K4rY_M3K4X
//     PlcTask Inputs/Main.M12.nRawEncoderULINT <-> FB Inputs Channel 2/Position
//     PlcTask Inputs/Main.M9.nRawEncoderULINT <-> FB Inputs Channel 1/Position
//   tmo_optics Instance <-> Device 1 (EtherCAT)/Term 1 (EK1200)/Term 5 (EK1122)/Term 20 (EK1100)/EL5042_M3K4Y_M3K4rX
//     PlcTask Inputs/Main.M13.nRawEncoderULINT <-> FB Inputs Channel 1/Position
//     PlcTask Inputs/Main.M14.nRawEncoderULINT <-> FB Inputs Channel 2/Position
//   tmo_optics Instance <-> Device 1 (EtherCAT)/Term 1 (EK1200)/Term 5 (EK1122)/Term 20 (EK1100)/EL5042_M3K4_BEND_USDS
//     PlcTask Inputs/Main.M15.nRawEncoderULINT <-> FB Inputs Channel 1/Position
//   tmo_optics Instance <-> Device 1 (EtherCAT)/Term 1 (EK1200)/Term 5 (EK1122)/Term 20 (EK1100)/EL7041-0052_M2K4X
//     PlcTask Inputs/Main.M7.bLimitBackwardEnable <-> STM Status/Status/Digital input 2
//     PlcTask Inputs/Main.M7.bLimitForwardEnable <-> STM Status/Status/Digital input 1
//   tmo_optics Instance <-> Device 1 (EtherCAT)/Term 1 (EK1200)/Term 5 (EK1122)/Term 20 (EK1100)/EL7041-0052_M2K4Y
//     PlcTask Inputs/Main.M8.bLimitBackwardEnable <-> STM Status/Status/Digital input 2
//     PlcTask Inputs/Main.M8.bLimitForwardEnable <-> STM Status/Status/Digital input 1
//   tmo_optics Instance <-> Device 1 (EtherCAT)/Term 1 (EK1200)/Term 5 (EK1122)/Term 20 (EK1100)/EL7041-0052_M2K4rY
//     PlcTask Inputs/Main.M9.bLimitBackwardEnable <-> STM Status/Status/Digital input 2
//     PlcTask Inputs/Main.M9.bLimitForwardEnable <-> STM Status/Status/Digital input 1
//   tmo_optics Instance <-> Device 1 (EtherCAT)/Term 1 (EK1200)/Term 5 (EK1122)/Term 20 (EK1100)/EL7041-0052_M3K4X
//     PlcTask Inputs/Main.M12.bLimitBackwardEnable <-> STM Status/Status/Digital input 2
//     PlcTask Inputs/Main.M12.bLimitForwardEnable <-> STM Status/Status/Digital input 1
//   tmo_optics Instance <-> Device 1 (EtherCAT)/Term 1 (EK1200)/Term 5 (EK1122)/Term 20 (EK1100)/EL7041-0052_M3K4Y
//     PlcTask Inputs/Main.M13.bLimitBackwardEnable <-> STM Status/Status/Digital input 2
//     PlcTask Inputs/Main.M13.bLimitForwardEnable <-> STM Status/Status/Digital input 1
//   tmo_optics Instance <-> Device 1 (EtherCAT)/Term 1 (EK1200)/Term 5 (EK1122)/Term 20 (EK1100)/EL7041-0052_M3K4rX
//     PlcTask Inputs/Main.M14.bLimitBackwardEnable <-> STM Status/Status/Digital input 2
//     PlcTask Inputs/Main.M14.bLimitForwardEnable <-> STM Status/Status/Digital input 1
//   tmo_optics Instance <-> Device 1 (EtherCAT)/Term 1 (EK1200)/Term 5 (EK1122)/Term 20 (EK1100)/EL7041_M2K4_BEND_DS
//     PlcTask Inputs/Main.M11.bLimitBackwardEnable <-> STM Status/Status/Digital input 2
//     PlcTask Inputs/Main.M11.bLimitForwardEnable <-> STM Status/Status/Digital input 1
//   tmo_optics Instance <-> Device 1 (EtherCAT)/Term 1 (EK1200)/Term 5 (EK1122)/Term 20 (EK1100)/EL7041_M2K4_BEND_US
//     PlcTask Inputs/Main.M10.bLimitBackwardEnable <-> STM Status/Status/Digital input 2
//     PlcTask Inputs/Main.M10.bLimitForwardEnable <-> STM Status/Status/Digital input 1
//   tmo_optics Instance <-> Device 1 (EtherCAT)/Term 1 (EK1200)/Term 5 (EK1122)/Term 20 (EK1100)/EL7041_M3K4_BEND_DS
//     PlcTask Inputs/Main.M16.bLimitBackwardEnable <-> STM Status/Status/Digital input 2
//     PlcTask Inputs/Main.M16.bLimitForwardEnable <-> STM Status/Status/Digital input 1
//   tmo_optics Instance <-> Device 1 (EtherCAT)/Term 1 (EK1200)/Term 5 (EK1122)/Term 20 (EK1100)/EL7041_M3K4_BEND_US
//     PlcTask Inputs/Main.M15.bLimitBackwardEnable <-> STM Status/Status/Digital input 2
//     PlcTask Inputs/Main.M15.bLimitForwardEnable <-> STM Status/Status/Digital input 1
//   tmo_optics Instance <-> Device 1 (EtherCAT)/Term 1 (EK1200)/Term 5 (EK1122)/Term 40 (EK1100)/EL3054_FWM_PRSM
//     PlcTask Inputs/PRG_MR2K4_KBO.fbCoolingPanel.fbFlow_1.iRaw <-> AI Standard Channel 1/Value
//     PlcTask Inputs/PRG_MR3K4_KBO.fbCoolingPanel.fbFlow_1.iRaw <-> AI Standard Channel 2/Value
//     PlcTask Inputs/PRG_MR2K4_KBO.fbCoolingPanel.fbPress_1.iRaw <-> AI Standard Channel 3/Value
//     PlcTask Inputs/PRG_MR3K4_KBO.fbCoolingPanel.fbPress_1.iRaw <-> AI Standard Channel 3/Value
//   tmo_optics Instance <-> Device 1 (EtherCAT)/Term 1 (EK1200)/Term 5 (EK1122)/Term 40 (EK1100)/EL3202-0010_M2K4DS2_M2K4DS3
//     PlcTask Inputs/GVL_M2K4_RTD.nM2K4DS_RTD_3 <-> RTD Inputs Channel 2/Value
//     PlcTask Inputs/PRG_MR2K4_KBO.fbM2K4_Chin_Right_RTD.bError <-> RTD Inputs Channel 1/Status/Error
//     PlcTask Inputs/PRG_MR2K4_KBO.fbM2K4_Chin_Right_RTD.bOverrange <-> RTD Inputs Channel 1/Status/Overrange
//     PlcTask Inputs/PRG_MR2K4_KBO.fbM2K4_Chin_Right_RTD.bUnderrange <-> RTD Inputs Channel 1/Status/Underrange
//     PlcTask Inputs/PRG_MR2K4_KBO.fbM2K4_Chin_Right_RTD.iRaw <-> RTD Inputs Channel 1/Value
//     PlcTask Inputs/P_StripeProtections.fbStripProtMR2K4.ffLowerCoatingRTemp.bError <-> RTD Inputs Channel 1/Status/Error
//     PlcTask Inputs/P_StripeProtections.fbStripProtMR2K4.ffLowerCoatingRTemp.bOverrange <-> RTD Inputs Channel 1/Status/Overrange
//     PlcTask Inputs/P_StripeProtections.fbStripProtMR2K4.ffLowerCoatingRTemp.bUnderrange <-> RTD Inputs Channel 1/Status/Underrange
//     PlcTask Inputs/P_StripeProtections.fbStripProtMR2K4.ffLowerCoatingRTemp.iRaw <-> RTD Inputs Channel 1/Value
//     PlcTask Inputs/P_StripeProtections.fbStripProtMR2K4.ffUpperCoatingRTemp.bError <-> RTD Inputs Channel 1/Status/Error
//     PlcTask Inputs/P_StripeProtections.fbStripProtMR2K4.ffUpperCoatingRTemp.bOverrange <-> RTD Inputs Channel 1/Status/Overrange
//     PlcTask Inputs/P_StripeProtections.fbStripProtMR2K4.ffUpperCoatingRTemp.bUnderrange <-> RTD Inputs Channel 1/Status/Underrange
//     PlcTask Inputs/P_StripeProtections.fbStripProtMR2K4.ffUpperCoatingRTemp.iRaw <-> RTD Inputs Channel 1/Value
//   tmo_optics Instance <-> Device 1 (EtherCAT)/Term 1 (EK1200)/Term 5 (EK1122)/Term 40 (EK1100)/EL3202-0010_M2K4US1_M2K4US2
//     PlcTask Inputs/GVL_M2K4_RTD.nM2K4US_RTD_1 <-> RTD Inputs Channel 1/Value
//     PlcTask Inputs/PRG_MR2K4_KBO.fbM2K4_Chin_Left_RTD.bError <-> RTD Inputs Channel 2/Status/Error
//     PlcTask Inputs/PRG_MR2K4_KBO.fbM2K4_Chin_Left_RTD.bOverrange <-> RTD Inputs Channel 2/Status/Overrange
//     PlcTask Inputs/PRG_MR2K4_KBO.fbM2K4_Chin_Left_RTD.bUnderrange <-> RTD Inputs Channel 2/Status/Underrange
//     PlcTask Inputs/PRG_MR2K4_KBO.fbM2K4_Chin_Left_RTD.iRaw <-> RTD Inputs Channel 2/Value
//     PlcTask Inputs/P_StripeProtections.fbStripProtMR2K4.ffLowerCoatingLTemp.bError <-> RTD Inputs Channel 2/Status/Error
//     PlcTask Inputs/P_StripeProtections.fbStripProtMR2K4.ffLowerCoatingLTemp.bOverrange <-> RTD Inputs Channel 2/Status/Overrange
//     PlcTask Inputs/P_StripeProtections.fbStripProtMR2K4.ffLowerCoatingLTemp.bUnderrange <-> RTD Inputs Channel 2/Status/Underrange
//     PlcTask Inputs/P_StripeProtections.fbStripProtMR2K4.ffLowerCoatingLTemp.iRaw <-> RTD Inputs Channel 2/Value
//     PlcTask Inputs/P_StripeProtections.fbStripProtMR2K4.ffUpperCoatingLTemp.bError <-> RTD Inputs Channel 2/Status/Error
//     PlcTask Inputs/P_StripeProtections.fbStripProtMR2K4.ffUpperCoatingLTemp.bOverrange <-> RTD Inputs Channel 2/Status/Overrange
//     PlcTask Inputs/P_StripeProtections.fbStripProtMR2K4.ffUpperCoatingLTemp.bUnderrange <-> RTD Inputs Channel 2/Status/Underrange
//     PlcTask Inputs/P_StripeProtections.fbStripProtMR2K4.ffUpperCoatingLTemp.iRaw <-> RTD Inputs Channel 2/Value
//   tmo_optics Instance <-> Device 1 (EtherCAT)/Term 1 (EK1200)/Term 5 (EK1122)/Term 40 (EK1100)/EL3202-0010_M2K4US3_M2K4DS1
//     PlcTask Inputs/GVL_M2K4_RTD.nM2K4DS_RTD_1 <-> RTD Inputs Channel 2/Value
//     PlcTask Inputs/GVL_M2K4_RTD.nM2K4US_RTD_3 <-> RTD Inputs Channel 1/Value
//   tmo_optics Instance <-> Device 1 (EtherCAT)/Term 1 (EK1200)/Term 5 (EK1122)/Term 40 (EK1100)/EL3202-0010_M3K4DS2_M3K4DS3
//     PlcTask Inputs/GVL_M3K4_RTD.nM3K4DS_RTD_3 <-> RTD Inputs Channel 2/Value
//     PlcTask Inputs/PRG_MR3K4_KBO.fbM3K4_Chin_Right_RTD.bError <-> RTD Inputs Channel 1/Status/Error
//     PlcTask Inputs/PRG_MR3K4_KBO.fbM3K4_Chin_Right_RTD.bOverrange <-> RTD Inputs Channel 1/Status/Overrange
//     PlcTask Inputs/PRG_MR3K4_KBO.fbM3K4_Chin_Right_RTD.bUnderrange <-> RTD Inputs Channel 1/Status/Underrange
//     PlcTask Inputs/PRG_MR3K4_KBO.fbM3K4_Chin_Right_RTD.iRaw <-> RTD Inputs Channel 1/Value
//     PlcTask Inputs/P_StripeProtections.fbStripProtMR3K4.ffLowerCoatingRTemp.bError <-> RTD Inputs Channel 1/Status/Error
//     PlcTask Inputs/P_StripeProtections.fbStripProtMR3K4.ffLowerCoatingRTemp.bOverrange <-> RTD Inputs Channel 1/Status/Overrange
//     PlcTask Inputs/P_StripeProtections.fbStripProtMR3K4.ffLowerCoatingRTemp.bUnderrange <-> RTD Inputs Channel 1/Status/Underrange
//     PlcTask Inputs/P_StripeProtections.fbStripProtMR3K4.ffLowerCoatingRTemp.iRaw <-> RTD Inputs Channel 1/Value
//     PlcTask Inputs/P_StripeProtections.fbStripProtMR3K4.ffUpperCoatingRTemp.bError <-> RTD Inputs Channel 1/Status/Error
//     PlcTask Inputs/P_StripeProtections.fbStripProtMR3K4.ffUpperCoatingRTemp.bOverrange <-> RTD Inputs Channel 1/Status/Overrange
//     PlcTask Inputs/P_StripeProtections.fbStripProtMR3K4.ffUpperCoatingRTemp.bUnderrange <-> RTD Inputs Channel 1/Status/Underrange
//     PlcTask Inputs/P_StripeProtections.fbStripProtMR3K4.ffUpperCoatingRTemp.iRaw <-> RTD Inputs Channel 1/Value
//   tmo_optics Instance <-> Device 1 (EtherCAT)/Term 1 (EK1200)/Term 5 (EK1122)/Term 40 (EK1100)/EL3202-0010_M3K4US1_M3K4US2
//     PlcTask Inputs/GVL_M3K4_RTD.nM3K4US_RTD_1 <-> RTD Inputs Channel 1/Value
//     PlcTask Inputs/PRG_MR3K4_KBO.fbM3K4_Chin_Left_RTD.bError <-> RTD Inputs Channel 2/Status/Error
//     PlcTask Inputs/PRG_MR3K4_KBO.fbM3K4_Chin_Left_RTD.bOverrange <-> RTD Inputs Channel 2/Status/Overrange
//     PlcTask Inputs/PRG_MR3K4_KBO.fbM3K4_Chin_Left_RTD.bUnderrange <-> RTD Inputs Channel 2/Status/Underrange
//     PlcTask Inputs/PRG_MR3K4_KBO.fbM3K4_Chin_Left_RTD.iRaw <-> RTD Inputs Channel 2/Value
//     PlcTask Inputs/P_StripeProtections.fbStripProtMR3K4.ffLowerCoatingLTemp.bError <-> RTD Inputs Channel 2/Status/Error
//     PlcTask Inputs/P_StripeProtections.fbStripProtMR3K4.ffLowerCoatingLTemp.bOverrange <-> RTD Inputs Channel 2/Status/Overrange
//     PlcTask Inputs/P_StripeProtections.fbStripProtMR3K4.ffLowerCoatingLTemp.bUnderrange <-> RTD Inputs Channel 2/Status/Underrange
//     PlcTask Inputs/P_StripeProtections.fbStripProtMR3K4.ffLowerCoatingLTemp.iRaw <-> RTD Inputs Channel 2/Value
//     PlcTask Inputs/P_StripeProtections.fbStripProtMR3K4.ffUpperCoatingLTemp.bError <-> RTD Inputs Channel 2/Status/Error
//     PlcTask Inputs/P_StripeProtections.fbStripProtMR3K4.ffUpperCoatingLTemp.bOverrange <-> RTD Inputs Channel 2/Status/Overrange
//     PlcTask Inputs/P_StripeProtections.fbStripProtMR3K4.ffUpperCoatingLTemp.bUnderrange <-> RTD Inputs Channel 2/Status/Underrange
//     PlcTask Inputs/P_StripeProtections.fbStripProtMR3K4.ffUpperCoatingLTemp.iRaw <-> RTD Inputs Channel 2/Value
//   tmo_optics Instance <-> Device 1 (EtherCAT)/Term 1 (EK1200)/Term 5 (EK1122)/Term 40 (EK1100)/EL3202-0010_M3K4US3_M3K4DS1
//     PlcTask Inputs/GVL_M3K4_RTD.nM3K4DS_RTD_1 <-> RTD Inputs Channel 2/Value
//     PlcTask Inputs/GVL_M3K4_RTD.nM3K4US_RTD_3 <-> RTD Inputs Channel 1/Value
//   tmo_optics Instance <-> Device 1 (EtherCAT)/Term 1 (EK1200)/Term 5 (EK1122)/Term 6 (EK1100)/EL1004_M1K4_STO
//     PlcTask Inputs/Main.M1K4.fbRunHOMS.bSTOEnable1 <-> Channel 1/Input
//     PlcTask Inputs/Main.M1K4.fbRunHOMS.bSTOEnable2 <-> Channel 2/Input
//   tmo_optics Instance <-> Device 1 (EtherCAT)/Term 1 (EK1200)/Term 5 (EK1122)/Term 6 (EK1100)/EL3054_M1K4_FWM_PRSM
//     PlcTask Inputs/PRG_MR1K4_SOMS.fbCoolingPanel.fbFlow_1.iRaw <-> AI Standard Channel 1/Value
//     PlcTask Inputs/PRG_MR1K4_SOMS.fbCoolingPanel.fbFlow_2.iRaw <-> AI Standard Channel 2/Value
//     PlcTask Inputs/PRG_MR1K4_SOMS.fbCoolingPanel.fbPress_1.iRaw <-> AI Standard Channel 3/Value
//   tmo_optics Instance <-> Device 1 (EtherCAT)/Term 1 (EK1200)/Term 5 (EK1122)/Term 6 (EK1100)/EL5042_M1K4_PitchBender
//     PlcTask Inputs/GVL_M1K4.M1K4_Pitch.diEncCnt <-> FB Inputs Channel 1/Position
//   tmo_optics Instance <-> Device 1 (EtherCAT)/Term 1 (EK1200)/Term 5 (EK1122)/Term 6 (EK1100)/EL5042_M1K4_Xupdwn
//     PlcTask Inputs/Main.M1K4.fbRunHOMS.stXdwnEnc/Count <-> FB Inputs Channel 2/Position
//     PlcTask Inputs/Main.M1K4.fbRunHOMS.stXupEnc/Count <-> FB Inputs Channel 1/Position
//   tmo_optics Instance <-> Device 1 (EtherCAT)/Term 1 (EK1200)/Term 5 (EK1122)/Term 6 (EK1100)/EL5042_M1K4_Yupdwn
//     PlcTask Inputs/Main.M1K4.fbRunHOMS.stYdwnEnc/Count <-> FB Inputs Channel 2/Position
//     PlcTask Inputs/Main.M1K4.fbRunHOMS.stYupEnc/Count <-> FB Inputs Channel 1/Position
//   tmo_optics Instance <-> Device 1 (EtherCAT)/Term 1 (EK1200)/Term 5 (EK1122)/Term 6 (EK1100)/EL6001_M1K4_PitchFine
//     SerialIO Inputs/GVL_SerialIO.Serial_stComIn_M1K4/D[{0..21}] <-> COM Inputs/Data In {0..21}  (22 links)
//     SerialIO Inputs/GVL_SerialIO.Serial_stComIn_M1K4/Status <-> COM Inputs/Status
//     SerialIO Outputs/GVL_SerialIO.Serial_stComOut_M1K4/Ctrl <-> COM Outputs/Ctrl
//     SerialIO Outputs/GVL_SerialIO.Serial_stComOut_M1K4/D[{0..21}] <-> COM Outputs/Data Out {0..21}  (22 links)
//   tmo_optics Instance <-> Device 1 (EtherCAT)/Term 1 (EK1200)/Term 5 (EK1122)/Term 6 (EK1100)/EL7041-1000_M1K4_PitchCoarse
//     PlcTask Inputs/Main.M5.bLimitBackwardEnable <-> STM Status/Status/Digital input 2
//     PlcTask Inputs/Main.M5.bLimitForwardEnable <-> STM Status/Status/Digital input 1
//   tmo_optics Instance <-> Device 1 (EtherCAT)/Term 1 (EK1200)/Term 5 (EK1122)/Term 6 (EK1100)/EL7041-1000_M1K4_Xdwn
//     PlcTask Inputs/Main.M4.bLimitBackwardEnable <-> STM Status/Status/Digital input 2
//     PlcTask Inputs/Main.M4.bLimitForwardEnable <-> STM Status/Status/Digital input 1
//   tmo_optics Instance <-> Device 1 (EtherCAT)/Term 1 (EK1200)/Term 5 (EK1122)/Term 6 (EK1100)/EL7041-1000_M1K4_Xup
//     PlcTask Inputs/Main.M3.bLimitBackwardEnable <-> STM Status/Status/Digital input 2
//     PlcTask Inputs/Main.M3.bLimitForwardEnable <-> STM Status/Status/Digital input 1
//   tmo_optics Instance <-> Device 1 (EtherCAT)/Term 1 (EK1200)/Term 5 (EK1122)/Term 6 (EK1100)/EL7041-1000_M1K4_Ydwn
//     PlcTask Inputs/Main.M2.bLimitBackwardEnable <-> STM Status/Status/Digital input 2
//     PlcTask Inputs/Main.M2.bLimitForwardEnable <-> STM Status/Status/Digital input 1
//   tmo_optics Instance <-> Device 1 (EtherCAT)/Term 1 (EK1200)/Term 5 (EK1122)/Term 6 (EK1100)/EL7041-1000_M1K4_Yup
//     PlcTask Inputs/Main.M1.bLimitBackwardEnable <-> STM Status/Status/Digital input 2
//     PlcTask Inputs/Main.M1.bLimitForwardEnable <-> STM Status/Status/Digital input 1
//   tmo_optics Instance <-> NC-Task 1 SAF/Axes/M1K4-Pitch
//     PlcTask Inputs/Main.M5.Axis.NcToPlc <-> Outputs/ToPlc
//     PlcTask Outputs/Main.M5.Axis.PlcToNc <-> Inputs/FromPlc
//   tmo_optics Instance <-> NC-Task 1 SAF/Axes/M1K4-Xdwn
//     PlcTask Inputs/Main.M4.Axis.NcToPlc <-> Outputs/ToPlc
//     PlcTask Outputs/Main.M4.Axis.PlcToNc <-> Inputs/FromPlc
//   tmo_optics Instance <-> NC-Task 1 SAF/Axes/M1K4-Xup
//     PlcTask Inputs/Main.M3.Axis.NcToPlc <-> Outputs/ToPlc
//     PlcTask Outputs/Main.M3.Axis.PlcToNc <-> Inputs/FromPlc
//   tmo_optics Instance <-> NC-Task 1 SAF/Axes/M1K4-Ydwn
//     PlcTask Inputs/Main.M2.Axis.NcToPlc <-> Outputs/ToPlc
//     PlcTask Outputs/Main.M2.Axis.PlcToNc <-> Inputs/FromPlc
//   tmo_optics Instance <-> NC-Task 1 SAF/Axes/M1K4-Yup
//     PlcTask Inputs/Main.M1.Axis.NcToPlc <-> Outputs/ToPlc
//     PlcTask Outputs/Main.M1.Axis.PlcToNc <-> Inputs/FromPlc
//   tmo_optics Instance <-> NC-Task 1 SAF/Axes/M2K4-BEND-DS
//     PlcTask Inputs/Main.M11.Axis.NcToPlc <-> Outputs/ToPlc
//     PlcTask Outputs/Main.M11.Axis.PlcToNc <-> Inputs/FromPlc
//   tmo_optics Instance <-> NC-Task 1 SAF/Axes/M2K4-BEND-US
//     PlcTask Inputs/Main.M10.Axis.NcToPlc <-> Outputs/ToPlc
//     PlcTask Outputs/Main.M10.Axis.PlcToNc <-> Inputs/FromPlc
//   tmo_optics Instance <-> NC-Task 1 SAF/Axes/M2K4-X
//     PlcTask Inputs/Main.M7.Axis.NcToPlc <-> Outputs/ToPlc
//     PlcTask Outputs/Main.M7.Axis.PlcToNc <-> Inputs/FromPlc
//   tmo_optics Instance <-> NC-Task 1 SAF/Axes/M2K4-Y
//     PlcTask Inputs/Main.M8.Axis.NcToPlc <-> Outputs/ToPlc
//     PlcTask Outputs/Main.M8.Axis.PlcToNc <-> Inputs/FromPlc
//   tmo_optics Instance <-> NC-Task 1 SAF/Axes/M2K4-rY
//     PlcTask Inputs/Main.M9.Axis.NcToPlc <-> Outputs/ToPlc
//     PlcTask Outputs/Main.M9.Axis.PlcToNc <-> Inputs/FromPlc
//   tmo_optics Instance <-> NC-Task 1 SAF/Axes/M3K4-BEND-DS
//     PlcTask Inputs/Main.M16.Axis.NcToPlc <-> Outputs/ToPlc
//     PlcTask Outputs/Main.M16.Axis.PlcToNc <-> Inputs/FromPlc
//   tmo_optics Instance <-> NC-Task 1 SAF/Axes/M3K4-BEND-US
//     PlcTask Inputs/Main.M15.Axis.NcToPlc <-> Outputs/ToPlc
//     PlcTask Outputs/Main.M15.Axis.PlcToNc <-> Inputs/FromPlc
//   tmo_optics Instance <-> NC-Task 1 SAF/Axes/M3K4-X
//     PlcTask Inputs/Main.M12.Axis.NcToPlc <-> Outputs/ToPlc
//     PlcTask Outputs/Main.M12.Axis.PlcToNc <-> Inputs/FromPlc
//   tmo_optics Instance <-> NC-Task 1 SAF/Axes/M3K4-Y
//     PlcTask Inputs/Main.M13.Axis.NcToPlc <-> Outputs/ToPlc
//     PlcTask Outputs/Main.M13.Axis.PlcToNc <-> Inputs/FromPlc
//   tmo_optics Instance <-> NC-Task 1 SAF/Axes/M3K4-rX
//     PlcTask Inputs/Main.M14.Axis.NcToPlc <-> Outputs/ToPlc
//     PlcTask Outputs/Main.M14.Axis.PlcToNc <-> Inputs/FromPlc
//   tmo_optics Instance <-> NC-Task 1 SAF/Axes/M4K4 X
//     PlcTask Inputs/Main.M17.Axis.NcToPlc <-> Outputs/ToPlc
//     PlcTask Outputs/Main.M17.Axis.PlcToNc <-> Inputs/FromPlc
//   tmo_optics Instance <-> NC-Task 1 SAF/Axes/M4K4 Y
//     PlcTask Inputs/Main.M18.Axis.NcToPlc <-> Outputs/ToPlc
//     PlcTask Outputs/Main.M18.Axis.PlcToNc <-> Inputs/FromPlc
//   tmo_optics Instance <-> NC-Task 1 SAF/Axes/M4K4 Z
//     PlcTask Inputs/Main.M19.Axis.NcToPlc <-> Outputs/ToPlc
//     PlcTask Outputs/Main.M19.Axis.PlcToNc <-> Inputs/FromPlc
//   tmo_optics Instance <-> NC-Task 1 SAF/Axes/M4K4 rX
//     PlcTask Inputs/Main.M20.Axis.NcToPlc <-> Outputs/ToPlc
//     PlcTask Outputs/Main.M20.Axis.PlcToNc <-> Inputs/FromPlc
//   tmo_optics Instance <-> NC-Task 1 SAF/Axes/M5K4 X
//     PlcTask Inputs/Main.M21.Axis.NcToPlc <-> Outputs/ToPlc
//     PlcTask Outputs/Main.M21.Axis.PlcToNc <-> Inputs/FromPlc
//   tmo_optics Instance <-> NC-Task 1 SAF/Axes/M5K4 Y
//     PlcTask Inputs/Main.M22.Axis.NcToPlc <-> Outputs/ToPlc
//     PlcTask Outputs/Main.M22.Axis.PlcToNc <-> Inputs/FromPlc
//   tmo_optics Instance <-> NC-Task 1 SAF/Axes/M5K4 Z
//     PlcTask Inputs/Main.M23.Axis.NcToPlc <-> Outputs/ToPlc
//     PlcTask Outputs/Main.M23.Axis.PlcToNc <-> Inputs/FromPlc
//   tmo_optics Instance <-> NC-Task 1 SAF/Axes/M5K4 rY
//     PlcTask Inputs/Main.M24.Axis.NcToPlc <-> Outputs/ToPlc
//     PlcTask Outputs/Main.M24.Axis.PlcToNc <-> Inputs/FromPlc
//   tmo_optics Instance <-> NC-Task 1 SAF/Axes/SL2K4_BOTTOM
//     PlcTask Inputs/Main.M26.Axis.NcToPlc <-> Outputs/ToPlc
//     PlcTask Outputs/Main.M26.Axis.PlcToNc <-> Inputs/FromPlc
//     PlcTask Outputs/Main.nM26Position <-> Enc/Inputs/In/nDataIn1
//   tmo_optics Instance <-> NC-Task 1 SAF/Axes/SL2K4_NORTH
//     PlcTask Inputs/Main.M27.Axis.NcToPlc <-> Outputs/ToPlc
//     PlcTask Outputs/Main.M27.Axis.PlcToNc <-> Inputs/FromPlc
//     PlcTask Outputs/Main.nM27Position <-> Enc/Inputs/In/nDataIn1
//   tmo_optics Instance <-> NC-Task 1 SAF/Axes/SL2K4_SOUTH
//     PlcTask Inputs/Main.M28.Axis.NcToPlc <-> Outputs/ToPlc
//     PlcTask Outputs/Main.M28.Axis.PlcToNc <-> Inputs/FromPlc
//     PlcTask Outputs/Main.nM28Position <-> Enc/Inputs/In/nDataIn1
//   tmo_optics Instance <-> NC-Task 1 SAF/Axes/SL2K4_TOP
//     PlcTask Inputs/Main.M25.Axis.NcToPlc <-> Outputs/ToPlc
//     PlcTask Outputs/Main.M25.Axis.PlcToNc <-> Inputs/FromPlc
//     PlcTask Outputs/Main.nM25Position <-> Enc/Inputs/In/nDataIn1

// ---- DUTs/ENUM_Si_B4C_Coating_States.TcDUT
{attribute 'qualified only'}
TYPE ENUM_Si_B4C_Coating_States :
(
    Unknown := 0,
    Si := 1,
    B4C := 2
);
END_TYPE

// ---- DUTs/ENUM_Si_B4C_Coating_States_1D.TcDUT
{attribute 'qualified_only'}
{attribute 'strict'}
{attribute 'to_string'}
TYPE ENUM_Si_B4C_Coating_States_1D :
(
     Unknown := 0,
    Si := 1,
    B4C := 2
)UINT;
END_TYPE

// ---- GVLs/GVL_PMPS.TcGVL
{attribute 'qualified_only'}
VAR_GLOBAL
    // FFO for devices upstream of ST1K0 (M1K4)
    {attribute 'pytmc' := '
        pv: PLC:TMO:OPTICS:FFO:01
    '}
    {attribute 'TcLinkTo' := '.q_xFastFaultOut:=TIIB[PMPS_FFO]^Channel 1^Output'}
    g_FastFaultOutput1 : FB_HardwareFFOutput := (bAutoReset:=TRUE, i_sNetID:='172.21.92.73.1.1');
    // FFO for devices downstream of ST1K0 (TMO hutch optics)
    {attribute 'pytmc' := '
        pv: PLC:TMO:OPTICS:FFO:02
    '}
    {attribute 'TcLinkTo' := '.q_xFastFaultOut:=TIIB[PMPS_FFO]^Channel 2^Output'}
    g_FastFaultOutput2 : FB_HardwareFFOutput := (bAutoReset:=TRUE, i_sNetID:='172.21.92.73.1.1');
    //FFO for devices downstream of ST4K0
     {attribute 'pytmc' := '
        pv: PLC:TMO:OPTICS:FFO:03
    '}

    g_FastFaultOutput3 : FB_HardwareFFOutput := (bAutoReset:=TRUE, i_sNetID:='172.21.92.73.1.1');


    // Arbiter for devices upstream of ST1K0 (M1K4)
    {attribute 'pytmc' := '
        pv: PLC:TMO:OPTICS:ARB:01
    '}
    g_fbArbiter1 : FB_Arbiter(1);
    // Arbiter for devices downstream of ST1K0 (TMO hutch optics)
    {attribute 'pytmc' := '
        pv: PLC:TMO:OPTICS:ARB:02
    '}
    g_fbArbiter2 : FB_Arbiter(2);
END_VAR

// ---- POUs/Main.TcPOU
PROGRAM Main
VAR
// M1K4
    // Motors
        {attribute 'TcLinkTo' := '.bLimitForwardEnable:=TIIB[EL7041-1000_M1K4_Yup]^STM Status^Status^Digital input 1;
                                  .bLimitBackwardEnable:=TIIB[EL7041-1000_M1K4_Yup]^STM Status^Status^Digital input 2'}
        {attribute 'pytmc' := '
            pv: MR1K4:SOMS:MMS:YUP
        '}
        //PMPS State Stage; bPowerSelf:=False
        M1 : ST_MotionStage := (sName:='MR1K4-Coatings', fVelocity:=200.0, nEnableMode:=ENUM_StageEnableMode.ALWAYS, bPowerSelf:=FALSE); // M1K4 Yup
        fbMotionStage_m1 : FB_MotionStage;

        {attribute 'TcLinkTo' := '.bLimitForwardEnable:=TIIB[EL7041-1000_M1K4_Ydwn]^STM Status^Status^Digital input 1;
                                  .bLimitBackwardEnable:=TIIB[EL7041-1000_M1K4_Ydwn]^STM Status^Status^Digital input 2'}
        {attribute 'pytmc' := '
            pv: MR1K4:SOMS:MMS:YDWN
        '}
        M2 : ST_MotionStage := (fVelocity:=200.0, nEnableMode:=ENUM_StageEnableMode.ALWAYS, bPowerSelf:=TRUE); // M1K4 Ydwn
        fbMotionStage_m2 : FB_MotionStage;

        {attribute 'TcLinkTo' := '.bLimitForwardEnable:=TIIB[EL7041-1000_M1K4_Xup]^STM Status^Status^Digital input 1;
                                  .bLimitBackwardEnable:=TIIB[EL7041-1000_M1K4_Xup]^STM Status^Status^Digital input 2'}
        {attribute 'pytmc' := '
            pv: MR1K4:SOMS:MMS:XUP
        '}
        M3 : ST_MotionStage := (fVelocity:=1000.0, nEnableMode:=ENUM_StageEnableMode.ALWAYS, bPowerSelf:=TRUE); // M1K4 Xup
        fbMotionStage_m3 : FB_MotionStage;

        {attribute 'TcLinkTo' := '.bLimitForwardEnable:=TIIB[EL7041-1000_M1K4_Xdwn]^STM Status^Status^Digital input 1;
                                  .bLimitBackwardEnable:=TIIB[EL7041-1000_M1K4_Xdwn]^STM Status^Status^Digital input 2'}
        {attribute 'pytmc' := '
            pv: MR1K4:SOMS:MMS:XDWN
        '}
        M4 : ST_MotionStage := (fVelocity:=1000.0, nEnableMode:=ENUM_StageEnableMode.ALWAYS, bPowerSelf:=TRUE); // M1K4 Xdwn
        fbMotionStage_m4 : FB_MotionStage;

        {attribute 'TcLinkTo' := '.bLimitForwardEnable:=TIIB[EL7041-1000_M1K4_PitchCoarse]^STM Status^Status^Digital input 1;
                                  .bLimitBackwardEnable:=TIIB[EL7041-1000_M1K4_PitchCoarse]^STM Status^Status^Digital input 2'}
        {attribute 'pytmc' := '
            pv: MR1K4:SOMS:MMS:PITCH
        '}
        M5 : ST_MotionStage := (fVelocity := 150.0, bPowerSelf:=TRUE, nEnableMode:=ENUM_StageEnableMode.ALWAYS); // M1K4 Pitch Stepper
        fbMotionStage_m5 : FB_MotionStage;

(*        {attribute 'TcLinkTo' := '.bLimitForwardEnable:=TIIB[EL7041-1000_M1K4_Bender]^STM Status^Status^Digital input 1;
                                  .bLimitBackwardEnable:=TIIB[EL7041-1000_M1K4_Bender]^STM Status^Status^Digital input 2'}
        {attribute 'pytmc' := '
            pv: MR1K4:SOMS:MMS:BENDER
        '}
        M6 : ST_MotionStage := (fVelocity := 150.0, bPowerSelf:=TRUE); // M1K4 Bender
        fbMotionStage_m6 : FB_MotionStage;
*)

    {attribute 'TcLinkTo' := '.fbRunHOMS.bSTOEnable1:=TIIB[EL1004_M1K4_STO]^Channel 1^Input;
                              .fbRunHOMS.bSTOEnable2:=TIIB[EL1004_M1K4_STO]^Channel 2^Input;
                              .fbRunHOMS.stYupEnc.Count:=TIIB[EL5042_M1K4_Yupdwn]^FB Inputs Channel 1^Position;
                              .fbRunHOMS.stYdwnEnc.Count:=TIIB[EL5042_M1K4_Yupdwn]^FB Inputs Channel 2^Position;
                              .fbRunHOMS.stXupEnc.Count:=TIIB[EL5042_M1K4_Xupdwn]^FB Inputs Channel 1^Position;
                              .fbRunHOMS.stXdwnEnc.Count:=TIIB[EL5042_M1K4_Xupdwn]^FB Inputs Channel 2^Position'}
    {attribute 'pytmc' := '
        pv: MR1K4:SOMS
    '}
    M1K4 : DUT_HOMS;

    // Encoder Arrays/RMS Watch:
        {attribute 'pytmc' := '
            pv: MR1K4:SOMS:ENC:Y
        '}
        fbYRMSErrorM1K4 : FB_RMSWatch;
        fMaxYRMSErrorM1K4 : LREAL;
        fMinYRMSErrorM1K4 : LREAL;

        {attribute 'pytmc' := '
            pv: MR1K4:SOMS:ENC:X
        '}
        fbXRMSErrorM1K4 : FB_RMSWatch;
        fMaxXRMSErrorM1K4 : LREAL;
        fMinXRMSErrorM1K4 : LREAL;

        {attribute 'pytmc' := '
            pv: MR1K4:SOMS:ENC:PITCH
        '}
        fbPitchRMSErrorM1K4 : FB_RMSWatch;
        fMaxPitchRMSErrorM1K4 : LREAL;
        fMinPitchRMSErrorM1K4 : LREAL;

        {attribute 'pytmc' := '
            pv: MR1K4:SOMS:ENC:BENDER
        '}
        fbBenderRMSErrorM1K4 : FB_RMSWatch;
        fMaxBenderRMSErrorM1K4 : LREAL;
        fMinBenderRMSErrorM1K4 : LREAL;

    // Piezo Pitch Control
        //fbM1K4PitchControl : FB_PitchControl;
        //bM1K4PitchDone : BOOL;
        //bM1K4PitchBusy : BOOL;

    // Bender Control
        fbBenderM1K4 : FB_Bender;

    // Raw Encoder Counts
        {attribute 'pytmc' := '
            pv: MR1K4:SOMS:ENC:YUP:CNT
            field: EGU cnt
            io: i
        '}
        nEncCntYupM1K4 : UDINT;
        {attribute 'pytmc' := '
            pv: MR1K4:SOMS:ENC:YDWN:CNT
            field: EGU cnt
            io: i
        '}
        nEncCntYdwnM1K4 : UDINT;
        {attribute 'pytmc' := '
            pv: MR1K4:SOMS:ENC:XUP:CNT
            field: EGU cnt
            io: i
        '}
        nEncCntXupM1K4 : UDINT;
        {attribute 'pytmc' := '
            pv: MR1K4:SOMS:ENC:XDWN:CNT
            field: EGU cnt
            io: i
        '}
        nEncCntXdwnM1K4 : UDINT;
        {attribute 'pytmc' := '
            pv: MR1K4:SOMS:ENC:PITCH:CNT
            field: EGU cnt
            io: i
        '}
        nEncCntPitchM1K4 : UDINT;

    // Encoder Reference Values
        {attribute 'pytmc' := '
            pv: MR1K4:SOMS:ENC:YUP:REF
            field: EGU cnt
            io: i
        '}
        nEncRefYupM1K4 : UDINT;
        {attribute 'pytmc' := '
            pv: MR1K4:SOMS:ENC:YDWN:REF
            field: EGU cnt
            io: i
        '}
        nEncRefYdwnM1K4 : UDINT;
        {attribute 'pytmc' := '
            pv: MR1K4:SOMS:ENC:XUP:REF
            field: EGU cnt
            io: i
        '}
        nEncRefXupM1K4 : UDINT;
        {attribute 'pytmc' := '
            pv: MR1K4:SOMS:ENC:XDWN:REF
            field: EGU cnt
            io: i
        '}
        nEncRefXdwnM1K4 : UDINT;
        {attribute 'pytmc' := '
            pv: MR1K4:SOMS:ENC:PITCH:REF
            field: EGU cnt
            io: i
        '}
        nEncRefPitchM1K4 : UDINT;
        mcReadParameterPitchM1K4 : MC_ReadParameter;
        fEncRefPitchM1K4_urad : LREAL; // Current Pitch encoder offset in urad

    // Common
    fEncLeverArm_mm : LREAL := 513.0;

// LAMP KB Motors
    //MR2K4 X
        {attribute 'TcLinkTo' := '.bLimitForwardEnable :=TIIB[EL7041-0052_M2K4X]^STM Status^Status^Digital input 1;
                                  .bLimitBackwardEnable:=TIIB[EL7041-0052_M2K4X]^STM Status^Status^Digital input 2;
                                  .nRawEncoderULINT    := TIIB[EL5042_M2K4X_M2K4Y]^FB Inputs Channel 1^Position'}
        {attribute 'pytmc' := '
        pv: MR2K4:KBO:MMS:X
        '}
        M7 : ST_MotionStage := (nEnableMode:=ENUM_StageEnableMode.ALWAYS, bPowerSelf:=TRUE);
        fbMotionStage_m7 : FB_MotionStage;
    //MR2K4 Y
        {attribute 'TcLinkTo' := '.bLimitForwardEnable :=TIIB[EL7041-0052_M2K4Y]^STM Status^Status^Digital input 1;
                                  .bLimitBackwardEnable:=TIIB[EL7041-0052_M2K4Y]^STM Status^Status^Digital input 2;
                                  .nRawEncoderULINT    := TIIB[EL5042_M2K4X_M2K4Y]^FB Inputs Channel 2^Position'}
        {attribute 'pytmc' := '
        pv: MR2K4:KBO:MMS:Y
        '}
        //PMPS State Stage; bPowerSelf:=False
        M8 : ST_MotionStage := (sName:='MR2K4-Coatings', nEnableMode:=ENUM_StageEnableMode.ALWAYS, bPowerSelf:=FALSE);
        fbMotionStage_m8 : FB_MotionStage;
    //MR2K4 rY
        {attribute 'TcLinkTo' := '.bLimitForwardEnable :=TIIB[EL7041-0052_M2K4rY]^STM Status^Status^Digital input 1;
                                  .bLimitBackwardEnable:=TIIB[EL7041-0052_M2K4rY]^STM Status^Status^Digital input 2;
                                  .nRawEncoderULINT    := TIIB[EL5042_M2K4rY_M3K4X]^FB Inputs Channel 1^Position'}
        {attribute 'pytmc' := '
        pv: MR2K4:KBO:MMS:PITCH
        '}
        M9 : ST_MotionStage := (nEnableMode:=ENUM_StageEnableMode.ALWAYS, bPowerSelf:=TRUE);
        fbMotionStage_m9 : FB_MotionStage;
    //MR2K4 US BEND
        {attribute 'TcLinkTo' := '.bLimitForwardEnable :=TIIB[EL7041_M2K4_BEND_US]^STM Status^Status^Digital input 1;
                                  .bLimitBackwardEnable:=TIIB[EL7041_M2K4_BEND_US]^STM Status^Status^Digital input 2;
                                  .nRawEncoderULINT    := TIIB[EL5042_M2K4_BEND_USDS]^FB Inputs Channel 1^Position'}
        {attribute 'pytmc' := '
        pv: MR2K4:KBO:MMS:BEND:US
        '}
        M10 : ST_MotionStage := (nEnableMode:=ENUM_StageEnableMode.DURING_MOTION, bPowerSelf:=TRUE);
        fbMotionStage_m10 : FB_MotionStage;
    //MR2K4 DS BEND
        {attribute 'TcLinkTo' := '.bLimitForwardEnable :=TIIB[EL7041_M2K4_BEND_DS]^STM Status^Status^Digital input 1;
                                  .bLimitBackwardEnable:=TIIB[EL7041_M2K4_BEND_DS]^STM Status^Status^Digital input 2;
                                  .nRawEncoderULINT    := TIIB[EL5042_M2K4_BEND_USDS]^FB Inputs Channel 2^Position'}
        {attribute 'pytmc' := '
        pv: MR2K4:KBO:MMS:BEND:DS
        '}
        M11 : ST_MotionStage := (nEnableMode:=ENUM_StageEnableMode.DURING_MOTION, bPowerSelf:=TRUE);
        fbMotionStage_m11 : FB_MotionStage;
    //MR3K4 X
        {attribute 'TcLinkTo' := '.bLimitForwardEnable :=TIIB[EL7041-0052_M3K4X]^STM Status^Status^Digital input 1;
                                  .bLimitBackwardEnable:=TIIB[EL7041-0052_M3K4X]^STM Status^Status^Digital input 2;
                                  .nRawEncoderULINT    := TIIB[EL5042_M2K4rY_M3K4X]^FB Inputs Channel 2^Position'}
        {attribute 'pytmc' := '
        pv: MR3K4:KBO:MMS:X
        '}
        //PMPS State Stage; bPowerSelf:=False
        M12 : ST_MotionStage := (sName:='MR3K4-Coatings', nEnableMode:=ENUM_StageEnableMode.ALWAYS, bPowerSelf:=FALSE);
        fbMotionStage_m12 : FB_MotionStage;
    //MR3K4 Y
        {attribute 'TcLinkTo' := '.bLimitForwardEnable :=TIIB[EL7041-0052_M3K4Y]^STM Status^Status^Digital input 1;
                                  .bLimitBackwardEnable:=TIIB[EL7041-0052_M3K4Y]^STM Status^Status^Digital input 2;
                                  .nRawEncoderULINT    := TIIB[EL5042_M3K4Y_M3K4rX]^FB Inputs Channel 1^Position'}
        {attribute 'pytmc' := '
        pv: MR3K4:KBO:MMS:Y
        '}
        M13 : ST_MotionStage := (nEnableMode:=ENUM_StageEnableMode.ALWAYS, bPowerSelf:=TRUE);
        fbMotionStage_m13 : FB_MotionStage;
    //MR3K4 rX
        {attribute 'TcLinkTo' := '.bLimitForwardEnable :=TIIB[EL7041-0052_M3K4rX]^STM Status^Status^Digital input 1;
                                  .bLimitBackwardEnable:=TIIB[EL7041-0052_M3K4rX]^STM Status^Status^Digital input 2;
                                  .nRawEncoderULINT    := TIIB[EL5042_M3K4Y_M3K4rX]^FB Inputs Channel 2^Position'}
        {attribute 'pytmc' := '
        pv: MR3K4:KBO:MMS:PITCH
        '}
        M14 : ST_MotionStage := (nEnableMode:=ENUM_StageEnableMode.ALWAYS, bPowerSelf:=TRUE);
        fbMotionStage_m14 : FB_MotionStage;
    //MR3K4 US BEND
        {attribute 'TcLinkTo' := '.bLimitForwardEnable :=TIIB[EL7041_M3K4_BEND_US]^STM Status^Status^Digital input 1;
                                  .bLimitBackwardEnable:=TIIB[EL7041_M3K4_BEND_US]^STM Status^Status^Digital input 2;
                                  .nRawEncoderULINT    := TIIB[EL5042_M3K4_BEND_USDS]^FB Inputs Channel 1^Position'}
        {attribute 'pytmc' := '
        pv: MR3K4:KBO:MMS:BEND:US
        '}
        M15 : ST_MotionStage := (nEnableMode:=ENUM_StageEnableMode.DURING_MOTION, bPowerSelf:=TRUE);
        fbMotionStage_m15 : FB_MotionStage;
        //////////////////////////////////
    //MR3K4 DS BEND
        {attribute 'TcLinkTo' := '.bLimitForwardEnable :=TIIB[EL7041_M3K4_BEND_DS]^STM Status^Status^Digital input 1;
                                  .bLimitBackwardEnable:=TIIB[EL7041_M3K4_BEND_DS]^STM Status^Status^Digital input 2;
                                  .nRawEncoderULINT    := TIIB[EL5042_M2K4_BEND_USDS]^FB Inputs Channel 2^Position'}
        {attribute 'pytmc' := '
        pv: MR3K4:KBO:MMS:BEND:DS
        '}
        M16 : ST_MotionStage := (nEnableMode:=ENUM_StageEnableMode.DURING_MOTION, bPowerSelf:=TRUE);
        fbMotionStage_m16 : FB_MotionStage;
    //M4K4 X
        {attribute 'TcLinkTo' := '.bLimitForwardEnable:=TIIB[EL7041-0052_M4K4X]^STM Status^Status^Digital input 1;
                              .bLimitBackwardEnable:=TIIB[EL7041-0052_M4K4X]^STM Status^Status^Digital input 2;
                              .nRawEncoderULINT:=TIIB[EL5042_M4K4X_M4K4Y]^FB Inputs Channel 1^Position'}
        {attribute 'pytmc' := '
            pv: MR4K4:KBO:MMS:X
        '}
        M17 : ST_MotionStage := (nEnableMode:=ENUM_StageEnableMode.ALWAYS, bPowerSelf:=FALSE);
        fbMotionStageM17 : FB_MotionStage;
    //M4K4 Y
        {attribute 'TcLinkTo' := '.bLimitForwardEnable:=TIIB[EL7041-0052_M4K4Y]^STM Status^Status^Digital input 1;
                              .bLimitBackwardEnable:=TIIB[EL7041-0052_M4K4Y]^STM Status^Status^Digital input 2;
                              .nRawEncoderULINT:=TIIB[EL5042_M4K4X_M4K4Y]^FB Inputs Channel 2^Position'}
        {attribute 'pytmc' := '
            pv: MR4K4:KBO:MMS:Y
        '}
        M18 : ST_MotionStage := (nEnableMode:=ENUM_StageEnableMode.ALWAYS, bPowerSelf:=TRUE);
        fbMotionStageM18 : FB_MotionStage;
    //M4K4 Z
        {attribute 'TcLinkTo' := '.bLimitForwardEnable:=TIIB[EL7041-0052_M4K4Z]^STM Status^Status^Digital input 2;
                              .bLimitBackwardEnable:=TIIB[EL7041-0052_M4K4Z]^STM Status^Status^Digital input 1;
                              .nRawEncoderULINT:=TIIB[EL5042_M4K4Z_M4K4rX]^FB Inputs Channel 1^Position'}
        {attribute 'pytmc' := '
            pv: MR4K4:KBO:MMS:Z
        '}
        M19 : ST_MotionStage := (nEnableMode:=ENUM_StageEnableMode.ALWAYS, bPowerSelf:=TRUE);
        fbMotionStageM19 : FB_MotionStage;

    //M4K4 rX
        {attribute 'TcLinkTo' := '.bLimitForwardEnable:=TIIB[EL7041-0052_M4K4rX]^STM Status^Status^Digital input 1;
                              .bLimitBackwardEnable:=TIIB[EL7041-0052_M4K4rX]^STM Status^Status^Digital input 2;
                              .nRawEncoderULINT:=TIIB[EL5042_M4K4Z_M4K4rX]^FB Inputs Channel 2^Position'}
        {attribute 'pytmc' := '
            pv: MR4K4:KBO:MMS:PITCH
        '}
        M20 : ST_MotionStage := (nEnableMode:=ENUM_StageEnableMode.ALWAYS, bPowerSelf:=TRUE);
        fbMotionStageM20 : FB_MotionStage;
    //M5K4 X
        {attribute 'TcLinkTo' := '.bLimitForwardEnable:=TIIB[EL7041-0052_M5K4X]^STM Status^Status^Digital input 1;
                              .bLimitBackwardEnable:=TIIB[EL7041-0052_M5K4X]^STM Status^Status^Digital input 2;
                              .nRawEncoderULINT:=TIIB[EL5042_M5K4X_M5K4Y]^FB Inputs Channel 1^Position'}
        {attribute 'pytmc' := '
            pv: MR5K4:KBO:MMS:X
        '}
        M21 : ST_MotionStage := (nEnableMode:=ENUM_StageEnableMode.ALWAYS, bPowerSelf:=TRUE);
        fbMotionStageM21 : FB_MotionStage;
    //M5K4 Y
        {attribute 'TcLinkTo' := '.bLimitForwardEnable:=TIIB[EL7041-0052_M5K4Y]^STM Status^Status^Digital input 1;
                              .bLimitBackwardEnable:=TIIB[EL7041-0052_M5K4Y]^STM Status^Status^Digital input 2;
                              .nRawEncoderULINT:=TIIB[EL5042_M5K4X_M5K4Y]^FB Inputs Channel 2^Position'}
        {attribute 'pytmc' := '
            pv: MR5K4:KBO:MMS:Y
        '}
        M22 : ST_MotionStage := (nEnableMode:=ENUM_StageEnableMode.ALWAYS, bPowerSelf:=FALSE);
        fbMotionStageM22 : FB_MotionStage;
    //M5K4 Z
        {attribute 'TcLinkTo' := '.bLimitForwardEnable:=TIIB[EL7041-0052_M5K4Z]^STM Status^Status^Digital input 2;
                              .bLimitBackwardEnable:=TIIB[EL7041-0052_M5K4Z]^STM Status^Status^Digital input 1;
                              .nRawEncoderULINT:=TIIB[EL5042_M5K4Z_M5K4rY]^FB Inputs Channel 1^Position'}
        {attribute 'pytmc' := '
            pv: MR5K4:KBO:MMS:Z
        '}
        M23 : ST_MotionStage := (nEnableMode:=ENUM_StageEnableMode.ALWAYS, bPowerSelf:=TRUE);
        fbMotionStageM23 : FB_MotionStage;
    //M5K4 rY
        {attribute 'TcLinkTo' := '.bLimitForwardEnable:=TIIB[EL7041-0052_M5K4rY]^STM Status^Status^Digital input 1;
                              .bLimitBackwardEnable:=TIIB[EL7041-0052_M5K4rY]^STM Status^Status^Digital input 2;
                              .nRawEncoderULINT:=TIIB[EL5042_M5K4Z_M5K4rY]^FB Inputs Channel 2^Position'}
        {attribute 'pytmc' := '
            pv: MR5K4:KBO:MMS:PITCH
        '}
        M24 : ST_MotionStage := (nEnableMode:=ENUM_StageEnableMode.ALWAYS, bPowerSelf:=TRUE);
        fbMotionStageM24 : FB_MotionStage;

        // SL2K4-SCATTER: 4 Axes
        // In order to get LVDT linked to NC motion, you have to first link the IO in the NC to the stepper interface, then clear link  Axis->Inputs->In->nDataIn1->nDataIn1[0], then rebuild
        {attribute 'pytmc' := 'pv: SL2K4:SCATTER:MMS:TOP'}
        {attribute 'TcLinkTo' := '.nRawEncoderDINT      := TIIB[SL2K4-EL5072-E1]^IND Inputs Channel 1^Position'}
        M25: ST_MotionStage := (sName := 'SL2K4:SCATTER:MMS:TOP', nEnableMode:=ENUM_StageEnableMode.DURING_MOTION, bPowerSelf:=TRUE);
        {attribute 'pytmc' := 'pv: SL2K4:SCATTER:MMS:BOTTOM'}
        {attribute 'TcLinkTo' := '.nRawEncoderDINT      := TIIB[SL2K4-EL5072-E1]^IND Inputs Channel 2^Position'}
        M26: ST_MotionStage := (sName := 'SL2K4:SCATTER:MMS:BOTTOM', nEnableMode:=ENUM_StageEnableMode.DURING_MOTION, bPowerSelf:=TRUE);
        {attribute 'pytmc' := 'pv: SL2K4:SCATTER:MMS:NORTH'}
        {attribute 'TcLinkTo' := '.nRawEncoderDINT      := TIIB[SL2K4-EL5072-E2]^IND Inputs Channel 1^Position'}
        M27: ST_MotionStage := (sName := 'SL2K4:SCATTER:MMS:NORTH', nEnableMode:=ENUM_StageEnableMode.DURING_MOTION, bPowerSelf:=TRUE);
        {attribute 'pytmc' := 'pv: SL2K4:SCATTER:MMS:SOUTH'}
        {attribute 'TcLinkTo' := '.nRawEncoderDINT      := TIIB[SL2K4-EL5072-E2]^IND Inputs Channel 2^Position'}
        M28: ST_MotionStage := (sName := 'SL2K4:SCATTER:MMS:SOUTH', nEnableMode:=ENUM_StageEnableMode.DURING_MOTION, bPowerSelf:=TRUE);

        fbMotionStage_m25: FB_MotionStage;
        fbMotionStage_m26: FB_MotionStage;
        fbMotionStage_m27: FB_MotionStage;
        fbMotionStage_m28: FB_MotionStage;

        {attribute 'TcLinkTo' := 'TINC^NC-Task 1 SAF^Axes^SL2K4_TOP^Enc^Inputs^In^nDataIn1'}
        nM25Position AT %Q*: UDINT;
        {attribute 'TcLinkTo' := 'TINC^NC-Task 1 SAF^Axes^SL2K4_BOTTOM^Enc^Inputs^In^nDataIn1'}
        nM26Position AT %Q*: UDINT;
        {attribute 'TcLinkTo' := 'TINC^NC-Task 1 SAF^Axes^SL2K4_NORTH^Enc^Inputs^In^nDataIn1'}
        nM27Position AT %Q*: UDINT;
        {attribute 'TcLinkTo' := 'TINC^NC-Task 1 SAF^Axes^SL2K4_SOUTH^Enc^Inputs^In^nDataIn1'}
        nM28Position AT %Q*: UDINT;

    //MR4K4 MR5K4 STO button
    {attribute 'TcLinkTo' := 'TIIB[Term 109 (EL1004)]^Channel 1^Input'}
    bDreamEnable1 AT %I* : BOOL;
        {attribute 'TcLinkTo' := 'TIIB[Term 109 (EL1004)]^Channel 2^Input'}
    bDreamEnable2 AT %I* : BOOL;
    // Encoder Arrays/RMS Watch:
        //MR2K4 X ENC RMS
        {attribute 'pytmc' := '
            pv: MR2K4:KBO:ENC:X
        '}
        fbXRMSErrorM2K4 : FB_RMSWatch;
        fMaxXRMSErrorM2K4 : LREAL;
        fMinXRMSErrorM2K4 : LREAL;
        //MR2K4 Y ENC RMS
        {attribute 'pytmc' := '
            pv: MR2K4:KBO:ENC:Y
        '}
        fbYRMSErrorM2K4 : FB_RMSWatch;
        fMaxYRMSErrorM2K4 : LREAL;
        fMinYRMSErrorM2K4 : LREAL;
        //MR2K4 rY ENC RMS
        {attribute 'pytmc' := '
            pv: MR2K4:KBO:ENC:PITCH
        '}
        fbrYRMSErrorM2K4 : FB_RMSWatch;
        fMaxrYRMSErrorM2K4 : LREAL;
        fMinrYRMSErrorM2K4 : LREAL;
        //MR2K4 US BENDER ENC RMS
        {attribute 'pytmc' := '
            pv: MR2K4:KBO:ENC:BEND:US
        '}
        fbBendUSRMSErrorM2K4 : FB_RMSWatch;
        fMaxBendUSRMSErrorM2K4 : LREAL;
        fMinBendUSRMSErrorM2K4 : LREAL;
        //MR2K4 DS BENDER ENC RMS
        {attribute 'pytmc' := '
            pv: MR2K4:KBO:ENC:BEND:DS
        '}
        fbBendDSRMSErrorM2K4 : FB_RMSWatch;
        fMaxBendDSRMSErrorM2K4 : LREAL;
        fMinBendDSRMSErrorM2K4 : LREAL;
        //MR3K4 X ENC RMS
        {attribute 'pytmc' := '
            pv: MR3K4:KBO:ENC:X
        '}
        fbXRMSErrorM3K4 : FB_RMSWatch;
        fMaxXRMSErrorM3K4 : LREAL;
        fMinXRMSErrorM3K4 : LREAL;
        //MR3K4 Y ENC RMS
        {attribute 'pytmc' := '
            pv: MR3K4:KBO:ENC:Y
        '}
        fbYRMSErrorM3K4 : FB_RMSWatch;
        fMaxYRMSErrorM3K4 : LREAL;
        fMinYRMSErrorM3K4 : LREAL;
        //MR3K4 rX ENC RMS
        {attribute 'pytmc' := '
            pv: MR3K4:KBO:ENC:PITCH
        '}
        fbrXRMSErrorM3K4 : FB_RMSWatch;
        fMaxrXRMSErrorM3K4 : LREAL;
        fMinrXRMSErrorM3K4 : LREAL;
        //MR3K4 US BENDER ENC RMS
        {attribute 'pytmc' := '
            pv: MR3K4:KBO:ENC:BEND:US
        '}
        fbBendUSRMSErrorM3K4 : FB_RMSWatch;
        fMaxBendUSRMSErrorM3K4 : LREAL;
        fMinBendUSRMSErrorM3K4 : LREAL;
        //MR3K4 DS BENDER ENC RMS
        {attribute 'pytmc' := '
            pv: MR3K4:KBO:ENC:BEND:DS
        '}
        fbBendDSRMSErrorM3K4 : FB_RMSWatch;
        fMaxBendDSRMSErrorM3K4 : LREAL;
        fMinBendDSRMSErrorM3K4 : LREAL;
        //MR4K4 X ENC RMS
        {attribute 'pytmc' := '
            pv: MR4K4:KBO:ENC:X
        '}
        fbXRMSErrorM4K4 : FB_RMSWatch;
        fMaxXRMSErrorM4K4 : LREAL;
        fMinXRMSErrorM4K4 : LREAL;

        //MR4K4 Y ENC RMS
        {attribute 'pytmc' := '
            pv: MR4K4:KBO:ENC:Y
        '}
        fbYRMSErrorM4K4 : FB_RMSWatch;
        fMaxYRMSErrorM4K4 : LREAL;
        fMinYRMSErrorM4K4 : LREAL;

        //MR4K4 Z ENC RMS
        {attribute 'pytmc' := '
            pv: MR4K4:KBO:ENC:Z
        '}
        fbZRMSErrorM4K4 : FB_RMSWatch;
        fMaxZRMSErrorM4K4 : LREAL;
        fMinZRMSErrorM4K4 : LREAL;
        //MR4K4 rX ENC RMS
        {attribute 'pytmc' := '
            pv: MR4K4:KBO:ENC:PITCH
        '}
        fbPRMSErrorM4K4 : FB_RMSWatch;
        fMaxPRMSErrorM4K4 : LREAL;
        fMinPRMSErrorM4K4 : LREAL;

        //MR5K4 X ENC RMS
        {attribute 'pytmc' := '
            pv: MR5K4:KBO:ENC:X
        '}
        fbXRMSErrorM5K4 : FB_RMSWatch;
        fMaxXRMSErrorM5K4 : LREAL;
        fMinXRMSErrorM5K4 : LREAL;

        //MR5K4 Y ENC RMS
        {attribute 'pytmc' := '
            pv: MR5K4:KBO:ENC:Y
        '}
        fbYRMSErrorM5K4 : FB_RMSWatch;
        fMaxYRMSErrorM5K4 : LREAL;
        fMinYRMSErrorM5K4 : LREAL;

        //MR5K4 Z ENC RMS
        {attribute 'pytmc' := '
            pv: MR5K4:KBO:ENC:Z
        '}
        fbZRMSErrorM5K4 : FB_RMSWatch;
        fMaxZRMSErrorM5K4 : LREAL;
        fMinZRMSErrorM5K4 : LREAL;
        //MR5K4 rX ENC RMS
        {attribute 'pytmc' := '
            pv: MR5K4:KBO:ENC:PITCH
        '}
        fbPRMSErrorM5K4 : FB_RMSWatch;
        fMaxPRMSErrorM5K4 : LREAL;
        fMinPRMSErrorM5K4 : LREAL;


    // Encoder Reference Values
        //MR2K4 X ENC REF
        {attribute 'pytmc' := '
            pv: MR2K4:KBO:ENC:X:REF
            field: EGU cnt
            io: i
        '}
        nEncRefXM2K4 : UDINT;
        //MR2K4 Y ENC REF
        {attribute 'pytmc' := '
            pv: MR2K4:KBO:ENC:Y:REF
            field: EGU cnt
            io: i
        '}
        nEncRefYM2K4 : UDINT;
        //MR2K4 rY ENC REF
        {attribute 'pytmc' := '
            pv: MR2K4:KBO:ENC:PITCH:REF
            field: EGU cnt
            io: i
        '}
        nEncRefrYM2K4 : UDINT;
        //MR3K4 X ENC REF
        {attribute 'pytmc' := '
            pv: MR3K4:KBO:ENC:X:REF
            field: EGU cnt
            io: i
        '}
        nEncRefXM3K4 : UDINT;
        //MR3K4 Y ENC REF
        {attribute 'pytmc' := '
            pv: MR3K4:KBO:ENC:Y:REF
            field: EGU cnt
            io: i
        '}
        nEncRefYM3K4 : UDINT;
        //MR3K4 rX ENC REF
        {attribute 'pytmc' := '
            pv: MR3K4:KBO:ENC:PITCH:REF
            field: EGU cnt
            io: i
        '}
        nEncRefrXM3K4 : UDINT;

    // Encoder raw counts
        //MR2K4 X ENC CNT
        {attribute 'pytmc' := '
            pv: MR2K4:KBO:ENC:X:CNT
            field: EGU cnt
            io: i
        '}
        nEncCntXM2K4 : UDINT;
        //MR2K4 Y ENC CNT
        {attribute 'pytmc' := '
            pv: MR2K4:KBO:ENC:Y:CNT
            field: EGU cnt
            io: i
        '}
        nEncCntYM2K4 : UDINT;
        //MR2K4 rY ENC CNT
        {attribute 'pytmc' := '
            pv: MR2K4:KBO:ENC:PITCH:CNT
            field: EGU cnt
            io: i
        '}
        nEncCntrYM2K4 : UDINT;
        //MR3K4 X ENC CNT
        {attribute 'pytmc' := '
            pv: MR3K4:KBO:ENC:X:CNT
            field: EGU cnt
            io: i
        '}
        nEncCntXM3K4 : UDINT;
        //MR3K4 Y ENC CNT
        {attribute 'pytmc' := '
            pv: MR3K4:KBO:ENC:Y:CNT
            field: EGU cnt
            io: i
        '}
        nEncCntYM3K4 : UDINT;
        //MR3K4 rX ENC CNT
        {attribute 'pytmc' := '
            pv: MR3K4:KBO:ENC:PITCH:CNT
            field: EGU cnt
            io: i
        '}
        nEncCntrXM3K4 : UDINT;

    //Emergency Stop for LAMP KBs (M2K4 and M3K4)
        LAMPbSTOEnable1 AT %I* : BOOL;
        LAMPbSTOEnable2 AT %I* : BOOL;

    // LAMP KB BENDER RTDs
    // M2K4 US RTDs
            {attribute 'pytmc' := '
                pv: MR2K4:KBO:RTD:BEND:US:1
                field: ASLO 0.1
                field: EGU C
                io: i
            '}
            fM2K4US_RTD_1 : REAL;
            {attribute 'pytmc' := '
                pv: MR2K4:KBO:RTD:BEND:US:3
                field: ASLO 0.1
                field: EGU C
                io: i
            '}
            fM2K4US_RTD_3 : REAL;

    // M2K4 DS RTDs
        {attribute 'pytmc' := '
            pv: MR2K4:KBO:RTD:BEND:DS:1
            field: ASLO 0.1
            field: EGU C
            io: i
        '}
        fM2K4DS_RTD_1 : REAL;
        {attribute 'pytmc' := '
            pv: MR2K4:KBO:RTD:BEND:DS:3
            field: ASLO 0.1
            field: EGU C
            io: i
        '}
        fM2K4DS_RTD_3 : REAL;
    // M3K4 US RTDs
        {attribute 'pytmc' := '
            pv: MR3K4:KBO:RTD:BEND:US:1
            field: ASLO 0.1
            field: EGU C
            io: i
        '}
        fM3K4US_RTD_1 : REAL;
        {attribute 'pytmc' := '
            pv: MR3K4:KBO:RTD:BEND:US:3
            field: ASLO 0.1
            field: EGU C
            io: i
        '}
        fM3K4US_RTD_3 : REAL;
    // M3K4 DS RTDs
        {attribute 'pytmc' := '
            pv: MR3K4:KBO:RTD:BEND:DS:1
            field: ASLO 0.1
            field: EGU C
            io: i
        '}
        fM3K4DS_RTD_1 : REAL;
        {attribute 'pytmc' := '
            pv: MR3K4:KBO:RTD:BEND:DS:3
            field: ASLO 0.1
            field: EGU cnt
            io: i
        '}
        fM3K4DS_RTD_3 AT %I* : REAL;

    // RTD error bit
        bM2K4US_RTD_1_Err AT %I*: BOOL;
        bM2K4US_RTD_2_Err AT %I*: BOOL;
        bM2K4US_RTD_3_Err AT %I*: BOOL;
        bM2K4DS_RTD_1_Err AT %I*: BOOL;
        bM2K4DS_RTD_2_Err AT %I*: BOOL;
        bM2K4DS_RTD_3_Err AT %I*: BOOL;
        bM3K4US_RTD_1_Err AT %I*: BOOL;
        bM3K4US_RTD_2_Err AT %I*: BOOL;
        bM3K4US_RTD_3_Err AT %I*: BOOL;
        bM3K4DS_RTD_1_Err AT %I*: BOOL;
        bM3K4DS_RTD_2_Err AT %I*: BOOL;
        bM3K4DS_RTD_3_Err AT %I*: BOOL;

// Logging
fbLogHandler : FB_LogHandler;


END_VAR

// M1K4
    M1K4.fbRunHOMS(stYup:=M1,
                   stYdwn:=M2,
                   stXup:=M3,
                   stXdwn:=M4,
                   stPitch:=M5,
                   nYupEncRef:=GVL_M1K4_Constants.nYUP_ENC_REF,
                   nYdwnEncRef:=GVL_M1K4_Constants.nYDWN_ENC_REF,
                   nXupEncRef:=GVL_M1K4_Constants.nXUP_ENC_REF,
                   nXdwnEncRef:=GVL_M1K4_Constants.nXDWN_ENC_REF,
                   bExecuteCoupleY:=M1K4.bExecuteCoupleY,
                   bExecuteCoupleX:=M1K4.bExecuteCoupleX,
                   bExecuteDecoupleY:=M1K4.bExecuteDecoupleY,
                   bExecuteDecoupleX:=M1K4.bExecuteDecoupleX,
                   bGantryAlreadyCoupledY=>M1K4.bGantryAlreadyCoupledY,
                   bGantryAlreadyCoupledX=>M1K4.bGantryAlreadyCoupledX,
                   nCurrGantryY=>M1K4.nCurrGantryY,
                   nCurrGantryX=>M1K4.nCurrGantryX);
(*    fbBenderM1K4(stBender:=M6,
                 bSTOEnable1:=M1K4.fbRunHOMS.bSTOEnable1,
                 bSTOEnable2:=M1K4.fbRunHOMS.bSTOEnable2);
*)
    // No slave motion through Epics
    M2.bExecute := FALSE; // M1K4-Ydwn
    M4.bExecute := FALSE; // M1K4-Xdwn

    // Convert nCurrGantry to um (smaller number) to read out in epics
        M1K4.fCurrGantryY_um := LINT_TO_REAL(M1K4.nCurrGantryY) / 1000.0;
        M1K4.fCurrGantryX_um := LINT_TO_REAL(M1K4.nCurrGantryX) / 1000.0;

    // FB_MotionStage's for non-piezo axes
        fbMotionStage_m1(stMotionStage:=M1);
        fbMotionStage_m2(stMotionStage:=M2);
        fbMotionStage_m3(stMotionStage:=M3);
        fbMotionStage_m4(stMotionStage:=M4);
        fbMotionStage_m5(stMotionStage:=M5);
//        fbMotionStage_m6(stMotionStage:=M6);

    // Calculate Pitch RMS Error:
        fbYRMSErrorM1K4(stMotionStage:=M1,
                        fMaxRMSError=>fMaxYRMSErrorM1K4,
                        fMinRMSError=>fMinYRMSErrorM1K4);

        fbXRMSErrorM1K4(stMotionStage:=M3,
                        fMaxRMSError=>fMaxXRMSErrorM1K4,
                        fMinRMSError=>fMinXRMSErrorM1K4);

        fbPitchRMSErrorM1K4(stMotionStage:=M5,
                            fMaxRMSError=>fMaxPitchRMSErrorM1K4,
                            fMinRMSError=>fMinPitchRMSErrorM1K4);

(*        fbBenderRMSErrorM1K4(stMotionStage:=M6,
                             fMaxRMSError=>fMaxBenderRMSErrorM1K4,
                             fMinRMSError=>fMinBenderRMSErrorM1K4);
*)
    // Pitch Control
        //fbM1K4PitchControl(Pitch:=GVL_M1K4.M1K4_Pitch,
                           //Stepper:=M5,
                           //lrCurrentSetpoint:=M5.fPosition,
                          //q_bDone=>bM1K4PitchDone,
                           //q_bBusy=>bM1K4PitchBusy);
    // When STO hit, need to reset SP
        //IF NOT M5.bHardwareEnable THEN
            //M5.fPosition := M5.stAxisStatus.fActPosition;
        //END_IF

    // Raw Encoder Counts For Epics
        nEncCntYupM1K4 := ULINT_TO_UDINT(M1K4.fbRunHOMS.stYupEnc.Count);
        nEncCntYdwnM1K4 := ULINT_TO_UDINT(M1K4.fbRunHOMS.stYdwnEnc.Count);
        nEncCntXupM1K4 := ULINT_TO_UDINT(M1K4.fbRunHOMS.stXupEnc.Count);
        nEncCntXdwnM1K4 := ULINT_TO_UDINT(M1K4.fbRunHOMS.stXdwnEnc.Count);
        nEncCntPitchM1K4 := LINT_TO_UDINT(GVL_M1K4.M1K4_Pitch.diEncCnt);

    // Encoder Reference Values For Epics
        nEncRefYupM1K4 := ULINT_TO_UDINT(GVL_M1K4_Constants.nYUP_ENC_REF);
        nEncRefYdwnM1K4 := ULINT_TO_UDINT(GVL_M1K4_Constants.nYDWN_ENC_REF);
        nEncRefXupM1K4 := ULINT_TO_UDINT(GVL_M1K4_Constants.nXUP_ENC_REF);
        nEncRefXdwnM1K4 := ULINT_TO_UDINT(GVL_M1K4_Constants.nXDWN_ENC_REF);
        mcReadParameterPitchM1K4(Axis:=M5.Axis,
                                 Enable:=TRUE,
                                 ParameterNumber:=MC_AxisParameter.AxisEncoderOffset,
                                 ReadMode:=READMODE_CYCLIC,
                                 Value=>fEncRefPitchM1K4_urad);

        nEncRefPitchM1K4 := LREAL_TO_UDINT(ABS(fEncRefPitchM1K4_urad) * fEncLeverArm_mm);
//////////////////////////////////////////////////////////
//M2K4 and M3K4
    //FB_Motion stages for LAMP KBs
        //MR2K4
            fbMotionStage_m7(stMotionStage:=M7);
            fbMotionStage_m8(stMotionStage:=M8);
            fbMotionStage_m9(stMotionStage:=M9);
        //MR2K4 BEND
            fbMotionStage_m10(stMotionStage:=M10);
            fbMotionStage_m11(stMotionStage:=M11);
        //MR3K4
            fbMotionStage_m12(stMotionStage:=M12);
            fbMotionStage_m13(stMotionStage:=M13);
            fbMotionStage_m14(stMotionStage:=M14);
        //MR3K4 BEND
            fbMotionStage_m15(stMotionStage:=M15);
            fbMotionStage_m16(stMotionStage:=M16);

//MR4K4 and MR5K4
            M17.bHardwareEnable := bDREAMEnable1 and bDREAMenable2;
            M18.bHardwareEnable := bDREAMEnable1 and bDREAMenable2;
            M19.bHardwareEnable := bDREAMEnable1 and bDREAMenable2;
            M20.bHardwareEnable := bDREAMEnable1 and bDREAMenable2;
            M21.bHardwareEnable := bDREAMEnable1 and bDREAMenable2;
            M22.bHardwareEnable := bDREAMEnable1 and bDREAMenable2;
            M23.bHardwareEnable := bDREAMEnable1 and bDREAMenable2;
            M24.bHardwareEnable := bDREAMEnable1 and bDREAMenable2;
        //MR4K4
            fbMotionStageM17(stMotionStage:=M17);
            fbMotionStageM18(stMotionStage:=M18);
            fbMotionStageM19(stMotionStage:=M19);
            fbMotionStageM20(stMotionStage:=M20);
        //MR5K4
            fbMotionStageM21(stMotionStage:=M21);
            fbMotionStageM22(stMotionStage:=M22);
            fbMotionStageM23(stMotionStage:=M23);
            fbMotionStageM24(stMotionStage:=M24);


    // Calculate Pitch RMS Error for LAMP KBs:
        //MR2K4 X ENC RMS
        fbXRMSErrorM2K4(stMotionStage:=M7,
                        fMaxRMSError=>fMaxXRMSErrorM2K4,
                        fMinRMSError=>fMinXRMSErrorM2K4);
        //MR2K4 Y ENC RMS
        fbYRMSErrorM2K4(stMotionStage:=M8,
                        fMaxRMSError=>fMaxYRMSErrorM2K4,
                        fMinRMSError=>fMinYRMSErrorM2K4);
        //MR2K4 rY ENC RMS
        fbrYRMSErrorM2K4(stMotionStage:=M9,
                        fMaxRMSError=>fMaxrYRMSErrorM2K4,
                        fMinRMSError=>fMinrYRMSErrorM2K4);
        //MR2K4 US BENDER ENC RMS
        fbBendUSRMSErrorM2K4(stMotionStage:=M10,
                             fMaxRMSError=>fMaxBendUSRMSErrorM2K4,
                             fMinRMSError=>fMinBendUSRMSErrorM2K4);
        //MR2K4 DS BENDER ENC RMS
        fbBendDSRMSErrorM2K4(stMotionStage:=M11,
                             fMaxRMSError=>fMaxBendDSRMSErrorM2K4,
                             fMinRMSError=>fMinBendDSRMSErrorM2K4);
        //MR3K4 X ENC RMS
        fbXRMSErrorM3K4(stMotionStage:=M12,
                        fMaxRMSError=>fMaxXRMSErrorM3K4,
                        fMinRMSError=>fMinXRMSErrorM3K4);
        //MR3K4 Y ENC RMS
        fbYRMSErrorM3K4(stMotionStage:=M13,
                        fMaxRMSError=>fMaxYRMSErrorM3K4,
                        fMinRMSError=>fMinYRMSErrorM3K4);
        //MR3K4 rX ENC RMS
        fbrXRMSErrorM3K4(stMotionStage:=M14,
                        fMaxRMSError=>fMaxrXRMSErrorM3K4,
                        fMinRMSError=>fMinrXRMSErrorM3K4);
        //MR3K4 US BENDER ENC RMS
        fbBendUSRMSErrorM3K4(stMotionStage:=M15,
                             fMaxRMSError=>fMaxBendUSRMSErrorM3K4,
                             fMinRMSError=>fMinBendUSRMSErrorM3K4);
        //MR3K4 DS BENDER ENC RMS
        fbBendDSRMSErrorM3K4(stMotionStage:=M16,
                             fMaxRMSError=>fMaxBendDSRMSErrorM3K4,
                             fMinRMSError=>fMinBendDSRMSErrorM3K4);
    // Calculate Pitch RMS Error for DREAM KBs:
        //MR4K4 X ENC RMS
        fbXRMSErrorM4K4(stMotionStage:=M17,
                        fMaxRMSError=>fMaxXRMSErrorM4K4,
                        fMinRMSError=>fMinXRMSErrorM4K4);
        //MR4K4 Y ENC RMS
        fbYRMSErrorM4K4(stMotionStage:=M18,
                        fMaxRMSError=>fMaxYRMSErrorM4K4,
                        fMinRMSError=>fMinYRMSErrorM4K4);
        //MR4K4 Z ENC RMS
        fbZRMSErrorM4K4(stMotionStage:=M19,
                        fMaxRMSError=>fMaxZRMSErrorM4K4,
                        fMinRMSError=>fMinZRMSErrorM4K4);
        //MR4K4 rX ENC RMS
        fbPRMSErrorM4K4(stMotionStage:=M20,
                        fMaxRMSError=>fMaxPRMSErrorM4K4,
                        fMinRMSError=>fMinPRMSErrorM4K4);
        //MR5K4 X ENC RMS
        fbXRMSErrorM5K4(stMotionStage:=M21,
                        fMaxRMSError=>fMaxXRMSErrorM5K4,
                        fMinRMSError=>fMinXRMSErrorM5K4);
        //MR5K4 Y ENC RMS
        fbYRMSErrorM5K4(stMotionStage:=M22,
                        fMaxRMSError=>fMaxYRMSErrorM5K4,
                        fMinRMSError=>fMinYRMSErrorM5K4);
        //MR5K4 Z ENC RMS
        fbZRMSErrorM5K4(stMotionStage:=M23,
                        fMaxRMSError=>fMaxZRMSErrorM5K4,
                        fMinRMSError=>fMinZRMSErrorM5K4);
        //MR5K4 rY ENC RMS
        fbPRMSErrorM5K4(stMotionStage:=M24,
                        fMaxRMSError=>fMaxPRMSErrorM5K4,
                        fMinRMSError=>fMinPRMSErrorM5K4);


    //STO for LAMP KBs
        //MR2K4
        M7.bHardwareEnable := LAMPbSTOEnable1 AND LAMPbSTOEnable2;
        M8.bHardwareEnable := LAMPbSTOEnable1 AND LAMPbSTOEnable2;
        M9.bHardwareEnable := LAMPbSTOEnable1 AND LAMPbSTOEnable2;
        //MR2K4 BEND
        M10.bHardwareEnable := LAMPbSTOEnable1 AND LAMPbSTOEnable2;
        M11.bHardwareEnable := LAMPbSTOEnable1 AND LAMPbSTOEnable2;
        //MR3K4
        M12.bHardwareEnable := LAMPbSTOEnable1 AND LAMPbSTOEnable2;
        M13.bHardwareEnable := LAMPbSTOEnable1 AND LAMPbSTOEnable2;
        M14.bHardwareEnable := LAMPbSTOEnable1 AND LAMPbSTOEnable2;
        //MR3K4 BEND
        M15.bHardwareEnable := LAMPbSTOEnable1 AND LAMPbSTOEnable2;
        M16.bHardwareEnable := LAMPbSTOEnable1 AND LAMPbSTOEnable2;

    // LAMP KB Encoder Reference Values For Epics
        nEncRefXM2K4  := ULINT_TO_UDINT(GVL_M2K4_Constants.nM2K4X_ENC_REF);
        nEncRefYM2K4  := ULINT_TO_UDINT(GVL_M2K4_Constants.nM2K4Y_ENC_REF);
        nEncRefrYM2K4 := ULINT_TO_UDINT(GVL_M2K4_Constants.nM2K4rY_ENC_REF);
        nEncRefXM3K4  := ULINT_TO_UDINT(GVL_M3K4_Constants.nM3K4X_ENC_REF);
        nEncRefYM3K4  := ULINT_TO_UDINT(GVL_M3K4_Constants.nM3K4Y_ENC_REF);
        nEncRefrXM3K4 := ULINT_TO_UDINT(GVL_M3K4_Constants.nM3K4rX_ENC_REF);

    // LAMP KB Encoder Count Values For Epics
        nEncCntXM2K4  := ULINT_TO_UDINT(M7.nRawEncoderULINT);
        nEncCntYM2K4  := ULINT_TO_UDINT(M8.nRawEncoderULINT);
        nEncCntrYM2K4 := ULINT_TO_UDINT(M9.nRawEncoderULINT);
        nEncCntXM3K4  := ULINT_TO_UDINT(M12.nRawEncoderULINT);
        nEncCntYM3K4  := ULINT_TO_UDINT(M13.nRawEncoderULINT);
        nEncCntrXM3K4 := ULINT_TO_UDINT(M14.nRawEncoderULINT);

;

    // LAMP KB Bender RTDs
        fM2K4US_RTD_1 := INT_TO_REAL(GVL_M2K4_RTD.nM2K4US_RTD_1);
        fM2K4US_RTD_3 := INT_TO_REAL(GVL_M2K4_RTD.nM2K4US_RTD_3);

        fM2K4DS_RTD_1 := INT_TO_REAL(GVL_M2K4_RTD.nM2K4DS_RTD_1);
        fM2K4DS_RTD_3 := INT_TO_REAL(GVL_M2K4_RTD.nM2K4DS_RTD_3);

        fM3K4US_RTD_1 := INT_TO_REAL(GVL_M3K4_RTD.nM3K4US_RTD_1);
        fM3K4US_RTD_3 := INT_TO_REAL(GVL_M3K4_RTD.nM3K4US_RTD_3);

        fM3K4DS_RTD_1 := INT_TO_REAL(GVL_M3K4_RTD.nM3K4DS_RTD_1);
        fM3K4DS_RTD_3 := INT_TO_REAL(GVL_M3K4_RTD.nM3K4DS_RTD_3);




    // RTD not connected if T=0
        bM2K4US_RTD_1_Err := fM2K4US_RTD_1 = 0;
        bM2K4US_RTD_3_Err := fM2K4US_RTD_3 = 0;
        bM2K4DS_RTD_1_Err := fM2K4DS_RTD_1 = 0;
        bM2K4DS_RTD_3_Err := fM2K4DS_RTD_3 = 0;

        bM3K4US_RTD_1_Err := fM3K4US_RTD_1 = 0;
        bM3K4US_RTD_3_Err := fM3K4US_RTD_3 = 0;
        bM3K4DS_RTD_1_Err := fM3K4DS_RTD_1 = 0;
        bM3K4DS_RTD_3_Err := fM3K4DS_RTD_3 = 0;

    // LAMP KB Bender RTD interlocks
        M10.bHardwareEnable R= fM2K4US_RTD_1 > 1000 OR bM2K4US_RTD_1_Err;
        M11.bHardwareEnable R= fM2K4DS_RTD_1 > 1000 OR bM2K4DS_RTD_1_Err;
        M15.bHardwareEnable R= fM3K4US_RTD_1 > 1000 OR bM3K4US_RTD_1_Err;
        M16.bHardwareEnable R= fM3K4DS_RTD_1 > 1000 OR bM3K4DS_RTD_1_Err;

    // SL2K4
    nM25Position := DINT_TO_UDINT(Main.M25.nRawEncoderDINT);

    Main.M25.bLimitBackwardEnable := TRUE;
    Main.M25.bLimitForwardEnable := TRUE;
    Main.M25.bHardwareEnable := TRUE;

    fbMotionStage_m25(stMotionStage:=Main.M25);

    nM26Position := DINT_TO_UDINT(Main.M26.nRawEncoderDINT);

    Main.M26.bLimitBackwardEnable := TRUE;
    Main.M26.bLimitForwardEnable := TRUE;
    Main.M26.bHardwareEnable := TRUE;

    fbMotionStage_m26(stMotionStage:=Main.M26);

    nM27Position := DINT_TO_UDINT(Main.M27.nRawEncoderDINT);

    Main.M27.bLimitBackwardEnable := TRUE;
    Main.M27.bLimitForwardEnable := TRUE;
    Main.M27.bHardwareEnable := TRUE;

    fbMotionStage_m27(stMotionStage:=Main.M27);

    nM28Position := DINT_TO_UDINT(Main.M28.nRawEncoderDINT);

    Main.M28.bLimitBackwardEnable := TRUE;
    Main.M28.bLimitForwardEnable := TRUE;
    Main.M28.bHardwareEnable := TRUE;

    fbMotionStage_m28(stMotionStage:=Main.M28);

// Environment
    PRG_Environment();
// States
    PRG_States();
// PMPS
    PRG_PMPS();
////////////////////////////////

// Logging
fbLogHandler();

END_PROGRAM

// ---- POUs/PRG_States.TcPOU
PROGRAM PRG_States
VAR
    {attribute 'pytmc' := '
     pv: MR1K4:SOMS:COATING:STATE;
     io: io;
    '}
    fbMR1K4_Coating_States: FB_Offset_Coating_States := (bBPOkAutoReset:= TRUE);

    {attribute 'pytmc' := '
     pv: MR2K4:KBO:COATING:STATE;
     io: io;
    '}
    fbMR2K4_Coating_States: FB_KBO_Coating_States := (bBPOkAutoReset:= TRUE);

    {attribute 'pytmc' := '
     pv: MR3K4:KBO:COATING:STATE;
     io: io;
    '}
    fbMR3K4_Coating_States: FB_KBO_Coating_States := (bBPOkAutoReset:= TRUE);



    {attribute 'pytmc' := '
     pv: MR4K4:KBO:COATING
     io: io
    '}
    fbMR4K4_Coating_States: FB_PositionStatePMPS1D;

    {attribute 'pytmc' := '
      pv: MR4K4:KBO:COATING:STATE:SET
      io: io
    '}
    eMR4K4StateSet:  ENUM_Si_B4C_Coating_States_1D;
    {attribute 'pytmc' := '
      pv: MR4K4:KBO:COATING:STATE:GET
      io: i
    '}
    eMR4K4StateGet:  ENUM_Si_B4C_Coating_States_1D;
    fbMR4K4XSetup: FB_StateSetupHelper;
    fbMR4K4Default: ST_PositionState := (
    fVelocity := 0.15,
    bUseRawCounts := TRUE,
    bMoveOk := TRUE,
    bValid := TRUE

    );
    aMR4K4CoatingStatesX: ARRAY[1..GeneralConstants.MAX_STATES] OF ST_PositionState;

    {attribute 'pytmc' := '
     pv: MR5K4:KBO:COATING
     io: io
    '}
    fbMR5K4_Coating_States: FB_PositionStatePMPS1D;
    {attribute 'pytmc' := '
      pv: MR5K4:KBO:COATING:STATE:SET
      io: io
    '}
    eMR5K4StateSet:  ENUM_Si_B4C_Coating_States_1D;
    {attribute 'pytmc' := '
      pv: MR5K4:KBO:COATING:STATE:GET
      io: i
    '}
    eMR5K4StateGet: ENUM_Si_B4C_Coating_States_1D;
    fbMR5K4YSetup: FB_StateSetupHelper;
    fbMR5K4Default: ST_PositionState := (
    fVelocity := 0.15,
    bUseRawCounts := TRUE,
    bMoveOK := TRUE,
    bValid := TRUE
    );

    aMR5K4CoatingStatesY: ARRAY[1..GeneralConstants.MAX_STATES] OF ST_PositionState;


  //  fbMR4K4_Coating_StatesX: INT;
END_VAR

//MR1K4 Coating States with PMPS
fbMR1K4_Coating_States.stCoating1.stPMPS.sPmpsState := 'MR1K4:SOMS-SILICON';
fbMR1K4_Coating_States.stCoating1.nEncoderCount := 22000532;

